C03652=1113.772,23.201,-52.779,179.827,6.837,149.312
C03653=1113.768,23.416,-52.792,179.828,6.841,149.313
C03654=1113.763,23.631,-52.805,179.828,6.845,149.313
C03655=1113.760,23.845,-52.819,179.829,6.848,149.314
C03656=1113.754,24.095,-52.833,179.830,6.853,149.315
C03657=1113.749,24.344,-52.848,179.831,6.857,149.315
C03658=1113.744,24.593,-52.864,179.832,6.861,149.316
C03659=1113.739,24.842,-52.879,179.833,6.866,149.317
C03660=1113.733,25.092,-52.894,179.833,6.869,149.317
C03661=1113.729,25.342,-52.909,179.834,6.874,149.318
C03662=1113.724,25.591,-52.925,179.835,6.878,149.319
C03663=1113.719,25.841,-52.940,179.836,6.883,149.320
C03664=1113.714,26.090,-52.955,179.837,6.887,149.320
C03665=1113.709,26.339,-52.971,179.838,6.891,149.321
C03666=1113.705,26.589,-52.986,179.838,6.895,149.322
C03667=1113.699,26.839,-53.001,179.839,6.900,149.322
C03668=1113.694,27.088,-53.016,179.840,6.904,149.323
C03669=1113.689,27.338,-53.032,179.841,6.908,149.324
C03670=1113.683,27.587,-53.047,179.842,6.913,149.324
C03671=1113.679,27.836,-53.062,179.843,6.917,149.325
C03672=1113.674,28.086,-53.078,179.844,6.922,149.326
C03673=1113.669,28.336,-53.094,179.844,6.925,149.327
C03674=1113.664,28.585,-53.109,179.845,6.929,149.327
C03675=1113.659,28.834,-53.124,179.846,6.934,149.328
C03676=1113.655,29.084,-53.140,179.847,6.938,149.329
C03677=1113.649,29.333,-53.155,179.848,6.943,149.329
C03678=1113.644,29.583,-53.171,179.849,6.947,149.330
C03679=1113.639,29.832,-53.186,179.849,6.951,149.331
C03680=1113.634,30.082,-53.202,179.850,6.955,149.331
C03681=1113.629,30.331,-53.218,179.851,6.959,149.332
C03682=1113.624,30.580,-53.233,179.852,6.964,149.333
C03683=1113.619,30.830,-53.248,179.853,6.968,149.334
C03684=1113.614,31.080,-53.264,179.854,6.973,149.334
C03685=1113.609,31.329,-53.280,179.855,6.976,149.335
C03686=1113.604,31.578,-53.295,179.856,6.980,149.336
C03687=1113.599,31.828,-53.310,179.857,6.985,149.336
C03688=1113.594,32.078,-53.326,179.858,6.989,149.337
C03689=1113.589,32.327,-53.341,179.859,6.993,149.338
C03690=1113.584,32.576,-53.357,179.860,6.998,149.338
C03691=1113.579,32.827,-53.373,179.860,7.001,149.339
C03692=1113.574,33.076,-53.388,179.861,7.005,149.339
C03693=1113.569,33.324,-53.404,179.862,7.010,149.340
C03694=1113.564,33.574,-53.420,179.864,7.014,149.341
C03695=1113.559,33.824,-53.436,179.865,7.018,149.341
C03696=1113.554,34.073,-53.451,179.866,7.023,149.342
C03697=1113.548,34.323,-53.467,179.866,7.026,149.343
C03698=1113.544,34.572,-53.482,179.867,7.030,149.343
C03699=1113.539,34.821,-53.498,179.868,7.035,149.344
C03700=1113.534,35.071,-53.514,179.869,7.039,149.345
C03701=1113.529,35.321,-53.530,179.870,7.043,149.345
C03702=1113.524,35.570,-53.546,179.871,7.048,149.346
C03703=1113.519,35.819,-53.561,179.872,7.051,149.347
C03704=1113.515,36.034,-53.574,179.873,7.056,149.347
C03705=1113.510,36.248,-53.588,179.874,7.059,149.348
C03706=1113.506,36.462,-53.602,179.874,7.062,149.348
C03707=1113.502,36.677,-53.615,179.875,7.066,149.349
C03708=1113.498,36.891,-53.629,179.876,7.070,149.350
C03709=1113.493,37.105,-53.643,179.877,7.073,149.350
C03710=1113.489,37.320,-53.656,179.878,7.076,149.351
C03711=1113.485,37.534,-53.670,179.879,7.081,149.351
C03712=1113.479,37.783,-53.686,179.879,7.084,149.352
C03713=1113.475,38.033,-53.702,179.881,7.088,149.352
C03714=1113.469,38.282,-53.718,179.882,7.092,149.353
C03715=1113.465,38.532,-53.733,179.883,7.097,149.354
C03716=1113.460,38.781,-53.750,179.884,7.101,149.354
C03717=1113.455,39.030,-53.765,179.885,7.105,149.355
C03718=1113.450,39.280,-53.781,179.885,7.109,149.356
C03719=1113.445,39.529,-53.798,179.887,7.113,149.356
C03720=1113.440,39.779,-53.814,179.888,7.117,149.357
C03721=1113.435,40.029,-53.829,179.889,7.122,149.358
C03722=1113.430,40.278,-53.846,179.890,7.126,149.358
C03723=1113.425,40.527,-53.861,179.891,7.130,149.359
C03724=1113.420,40.776,-53.878,179.892,7.133,149.359
C03725=1113.415,41.026,-53.894,179.893,7.138,149.360
C03726=1113.410,41.275,-53.910,179.894,7.142,149.361
C03727=1113.405,41.525,-53.926,179.895,7.146,149.361
C03728=1113.400,41.775,-53.941,179.896,7.150,149.362
C03729=1113.395,42.024,-53.958,179.898,7.155,149.362
C03730=1113.390,42.273,-53.974,179.898,7.158,149.363
C03731=1113.386,42.523,-53.990,179.899,7.162,149.364
C03732=1113.380,42.772,-54.006,179.900,7.167,149.364
C03733=1113.376,43.022,-54.023,179.902,7.171,149.365
C03734=1113.370,43.271,-54.038,179.903,7.175,149.365
C03735=1113.366,43.521,-54.055,179.903,7.178,149.366
C03736=1113.361,43.770,-54.071,179.904,7.183,149.367
C03737=1113.356,44.020,-54.087,179.905,7.187,149.367
C03738=1113.351,44.268,-54.103,179.907,7.191,149.368
C03739=1113.346,44.519,-54.119,179.908,7.195,149.368
C03740=1113.341,44.767,-54.136,179.909,7.200,149.369
C03741=1113.336,45.017,-54.152,179.910,7.203,149.370
C03742=1113.330,45.266,-54.169,179.911,7.207,149.370
C03743=1113.326,45.516,-54.185,179.912,7.211,149.371
C03744=1113.321,45.765,-54.201,179.913,7.216,149.371
C03745=1113.316,46.015,-54.217,179.914,7.220,149.372
C03746=1113.311,46.264,-54.234,179.916,7.224,149.373
C03747=1113.306,46.514,-54.250,179.916,7.227,149.373
C03748=1113.301,46.763,-54.266,179.917,7.232,149.374
C03749=1113.297,47.012,-54.283,179.919,7.236,149.374
C03750=1113.292,47.262,-54.299,179.920,7.240,149.375
C03751=1113.286,47.511,-54.316,179.921,7.244,149.376
C03752=1113.282,47.761,-54.332,179.923,7.248,149.376
C03753=1113.276,48.010,-54.348,179.923,7.252,149.377
C03754=1113.272,48.260,-54.364,179.924,7.256,149.377
C03755=1113.267,48.508,-54.381,179.925,7.260,149.378
C03756=1113.262,48.758,-54.397,179.927,7.264,149.378
C03757=1113.257,49.008,-54.414,179.928,7.268,149.379
C03758=1113.252,49.257,-54.430,179.929,7.271,149.379
C03759=1113.247,49.507,-54.447,179.930,7.276,149.380
C03760=1113.243,49.721,-54.461,179.932,7.280,149.381
C03761=1113.239,49.935,-54.475,179.932,7.283,149.381
C03762=1113.234,50.149,-54.489,179.933,7.286,149.382
C03763=1113.230,50.363,-54.504,179.934,7.289,149.382
C03764=1113.226,50.578,-54.518,179.935,7.293,149.383
C03765=1113.222,50.792,-54.532,179.936,7.297,149.383
C03766=1113.217,51.006,-54.547,179.937,7.300,149.384
C03767=1113.213,51.220,-54.561,179.938,7.304,149.384
C03768=1113.208,51.470,-54.577,179.939,7.308,149.385
C03769=1113.203,51.719,-54.593,179.940,7.311,149.385
C03770=1113.198,51.969,-54.611,179.941,7.316,149.386
C03771=1113.193,52.218,-54.627,179.943,7.320,149.386
C03772=1113.188,52.467,-54.644,179.944,7.324,149.387
C03773=1113.183,52.717,-54.661,179.945,7.328,149.388
C03774=1113.179,52.966,-54.677,179.947,7.332,149.388
C03775=1113.174,53.215,-54.694,179.947,7.336,149.389
C03776=1113.168,53.465,-54.711,179.948,7.340,149.389
C03777=1113.164,53.714,-54.728,179.950,7.344,149.390
C03778=1113.159,53.963,-54.744,179.951,7.348,149.390
C03779=1113.154,54.213,-54.761,179.953,7.352,149.391
C03780=1113.149,54.462,-54.778,179.954,7.356,149.391
C03781=1113.144,54.711,-54.794,179.955,7.359,149.392
C03782=1113.139,54.961,-54.812,179.956,7.364,149.392
C03783=1113.134,55.210,-54.828,179.957,7.368,149.393
C03784=1113.130,55.460,-54.845,179.958,7.372,149.394
C03785=1113.124,55.709,-54.862,179.960,7.376,149.394
C03786=1113.120,55.958,-54.878,179.961,7.380,149.395
C03787=1113.114,56.208,-54.896,179.961,7.384,149.395
C03788=1113.109,56.457,-54.912,179.963,7.388,149.396
C03789=1113.104,56.707,-54.929,179.964,7.392,149.396
C03790=1113.100,56.956,-54.946,179.966,7.396,149.397
C03791=1113.095,57.206,-54.963,179.967,7.400,149.397
C03792=1113.089,57.455,-54.980,179.968,7.404,149.398
C03793=1113.085,57.704,-54.996,179.969,7.408,149.399
C03794=1113.080,57.954,-55.013,179.970,7.411,149.399
C03795=1113.075,58.203,-55.031,179.971,7.416,149.400
C03796=1113.070,58.452,-55.048,179.973,7.420,149.400
C03797=1113.065,58.702,-55.064,179.974,7.424,149.401
C03798=1113.060,58.951,-55.082,179.976,7.428,149.401
C03799=1113.055,59.201,-55.098,179.977,7.432,149.402
C03800=1113.050,59.451,-55.116,179.978,7.436,149.402
C03801=1113.045,59.699,-55.133,179.979,7.439,149.403
C03802=1113.040,59.949,-55.150,179.980,7.443,149.403
C03803=1113.036,60.198,-55.167,179.982,7.447,149.404
C03804=1113.031,60.448,-55.184,179.983,7.452,149.404
C03805=1113.026,60.697,-55.201,179.985,7.456,149.405
C03806=1113.021,60.946,-55.218,179.986,7.460,149.405
C03807=1113.016,61.195,-55.235,179.987,7.464,149.406
C03808=1113.011,61.445,-55.252,179.988,7.467,149.407
C03809=1113.007,61.694,-55.269,179.989,7.471,149.407
C03810=1113.001,61.944,-55.287,179.991,7.475,149.407
C03811=1112.997,62.193,-55.303,179.992,7.479,149.408
C03812=1112.992,62.442,-55.321,179.994,7.483,149.409
C03813=1112.986,62.692,-55.338,179.995,7.488,149.409
C03814=1112.982,62.941,-55.355,179.996,7.491,149.410
C03815=1112.977,63.190,-55.373,179.997,7.495,149.410
C03816=1112.973,63.404,-55.387,179.998,7.499,149.411
C03817=1112.969,63.619,-55.403,179.999,7.502,149.411
C03818=1112.965,63.832,-55.417,-180.000,7.505,149.412
C03819=1112.960,64.047,-55.431,-179.998,7.509,149.412
C03820=1112.956,64.262,-55.447,-179.997,7.512,149.412
C03821=1112.952,64.475,-55.461,-179.996,7.515,149.413
C03822=1112.947,64.689,-55.476,-179.995,7.519,149.413
C03823=1112.943,64.904,-55.491,-179.994,7.522,149.414
C03824=1112.939,65.153,-55.509,-179.992,7.526,149.414
C03825=1112.933,65.403,-55.526,-179.991,7.530,149.415
C03826=1112.929,65.652,-55.544,-179.990,7.534,149.415
C03827=1112.924,65.901,-55.561,-179.988,7.538,149.416
C03828=1112.918,66.150,-55.579,-179.988,7.542,149.416
C03829=1112.914,66.399,-55.595,-179.986,7.546,149.417
C03830=1112.909,66.649,-55.613,-179.985,7.550,149.417
C03831=1112.904,66.898,-55.630,-179.983,7.554,149.418
C03832=1112.900,67.147,-55.648,-179.982,7.558,149.418
C03833=1112.894,67.397,-55.665,-179.981,7.562,149.419
C03834=1112.890,67.646,-55.683,-179.979,7.566,149.419
C03835=1112.884,67.896,-55.700,-179.978,7.570,149.420
C03836=1112.880,68.145,-55.718,-179.977,7.573,149.420
C03837=1112.875,68.395,-55.735,-179.975,7.577,149.421
C03838=1112.870,68.644,-55.753,-179.974,7.581,149.421
C03839=1112.865,68.893,-55.771,-179.973,7.585,149.422
C03840=1112.861,69.143,-55.788,-179.971,7.589,149.422
C03841=1112.856,69.392,-55.806,-179.970,7.593,149.423
C03842=1112.851,69.641,-55.824,-179.969,7.598,149.423
C03843=1112.846,69.891,-55.841,-179.967,7.601,149.424
C03844=1112.841,70.140,-55.859,-179.965,7.605,149.424
C03845=1112.836,70.389,-55.875,-179.964,7.610,149.425
C03846=1112.831,70.639,-55.893,-179.963,7.613,149.425
C03847=1112.826,70.888,-55.911,-179.962,7.617,149.426
C03848=1112.821,71.137,-55.929,-179.961,7.621,149.426
C03849=1112.816,71.387,-55.947,-179.959,7.625,149.427
C03850=1112.811,71.636,-55.965,-179.958,7.629,149.427
C03851=1112.807,71.885,-55.982,-179.956,7.633,149.428
C03852=1112.802,72.134,-55.999,-179.955,7.637,149.428
C03853=1112.797,72.384,-56.017,-179.953,7.641,149.429
C03854=1112.792,72.633,-56.035,-179.952,7.645,149.429
C03855=1112.787,72.882,-56.053,-179.951,7.649,149.430
C03856=1112.782,73.132,-56.071,-179.949,7.653,149.430
C03857=1112.777,73.381,-56.088,-179.948,7.656,149.431
C03858=1112.772,73.630,-56.106,-179.947,7.660,149.431
C03859=1112.767,73.879,-56.124,-179.945,7.664,149.432
C03860=1112.763,74.129,-56.143,-179.944,7.668,149.432
C03861=1112.759,74.378,-56.160,-179.942,7.672,149.433
C03862=1112.754,74.628,-56.177,-179.941,7.676,149.433
C03863=1112.749,74.877,-56.195,-179.939,7.680,149.434
C03864=1112.744,75.126,-56.213,-179.938,7.684,149.434
C03865=1112.739,75.375,-56.231,-179.937,7.688,149.435
C03866=1112.734,75.625,-56.249,-179.935,7.692,149.435
C03867=1112.729,75.874,-56.267,-179.934,7.696,149.436
C03868=1112.724,76.123,-56.285,-179.932,7.700,149.436
C03869=1112.719,76.372,-56.303,-179.931,7.704,149.437
C03870=1112.715,76.622,-56.322,-179.930,7.707,149.437
C03871=1112.710,76.872,-56.339,-179.928,7.711,149.438
C03872=1112.705,77.085,-56.355,-179.927,7.715,149.438
C03873=1112.701,77.300,-56.370,-179.927,7.718,149.439
C03874=1112.697,77.513,-56.386,-179.926,7.721,149.439
C03875=1112.693,77.728,-56.401,-179.925,7.724,149.440
C03876=1112.688,77.941,-56.417,-179.924,7.727,149.440
C03877=1112.685,78.156,-56.432,-179.923,7.730,149.441
C03878=1112.680,78.369,-56.447,-179.923,7.734,149.441
C03879=1112.676,78.584,-56.463,-179.922,7.737,149.442
C03880=1112.671,78.833,-56.481,-179.920,7.741,149.442
C03881=1112.666,79.082,-56.499,-179.920,7.744,149.443
C03882=1112.661,79.331,-56.517,-179.918,7.749,149.443
C03883=1112.656,79.582,-56.536,-179.917,7.752,149.444
C03884=1112.652,79.830,-56.554,-179.916,7.756,149.444
C03885=1112.647,80.079,-56.572,-179.915,7.759,149.445
C03886=1112.642,80.329,-56.590,-179.914,7.764,149.446
C03887=1112.637,80.578,-56.608,-179.913,7.767,149.446
C03888=1112.633,80.828,-56.627,-179.912,7.771,149.447
C03889=1112.628,81.077,-56.645,-179.911,7.774,149.447
C03890=1112.623,81.326,-56.663,-179.910,7.778,149.448
C03891=1112.618,81.575,-56.681,-179.909,7.781,149.448
C03892=1112.612,81.825,-56.699,-179.908,7.786,149.449
C03893=1112.608,82.075,-56.718,-179.906,7.790,149.449
C03894=1112.603,82.323,-56.736,-179.906,7.793,149.450
C03895=1112.599,82.572,-56.754,-179.904,7.797,149.450
C03896=1112.594,82.821,-56.772,-179.904,7.801,149.451
C03897=1112.589,83.071,-56.791,-179.902,7.804,149.451
C03898=1112.584,83.321,-56.809,-179.901,7.809,149.452
C03899=1112.579,83.569,-56.828,-179.900,7.812,149.452
C03900=1112.574,83.818,-56.846,-179.899,7.816,149.453
C03901=1112.570,84.068,-56.864,-179.898,7.819,149.453
C03902=1112.565,84.318,-56.882,-179.896,7.823,149.454
C03903=1112.560,84.567,-56.900,-179.895,7.827,149.455
C03904=1112.555,84.816,-56.919,-179.894,7.830,149.455
C03905=1112.550,85.065,-56.938,-179.893,7.835,149.456
C03906=1112.545,85.315,-56.956,-179.892,7.839,149.456
C03907=1112.540,85.564,-56.974,-179.891,7.842,149.457
C03908=1112.535,85.813,-56.993,-179.889,7.846,149.457
C03909=1112.531,86.063,-57.011,-179.888,7.850,149.458
C03910=1112.526,86.312,-57.029,-179.887,7.853,149.458
C03911=1112.521,86.560,-57.048,-179.886,7.857,149.459
C03912=1112.516,86.810,-57.067,-179.884,7.861,149.459
C03913=1112.511,87.060,-57.085,-179.884,7.865,149.460
C03914=1112.507,87.308,-57.104,-179.882,7.869,149.460
C03915=1112.502,87.558,-57.123,-179.881,7.872,149.461
C03916=1112.497,87.808,-57.141,-179.880,7.876,149.461
C03917=1112.492,88.056,-57.159,-179.878,7.880,149.462
C03918=1112.487,88.306,-57.178,-179.877,7.884,149.462
C03919=1112.483,88.555,-57.197,-179.876,7.888,149.463
C03920=1112.478,88.804,-57.215,-179.875,7.891,149.463
C03921=1112.473,89.054,-57.233,-179.873,7.895,149.464
C03922=1112.468,89.303,-57.252,-179.872,7.899,149.464
C03923=1112.463,89.552,-57.270,-179.870,7.903,149.465
C03924=1112.458,89.802,-57.290,-179.869,7.906,149.465
C03925=1112.453,90.051,-57.308,-179.868,7.911,149.466
C03926=1112.449,90.299,-57.327,-179.867,7.914,149.466
C03927=1112.444,90.549,-57.346,-179.865,7.918,149.467
C03928=1112.439,90.763,-57.361,-179.864,7.921,149.467
C03929=1112.436,90.977,-57.378,-179.863,7.925,149.468
C03930=1112.432,91.191,-57.394,-179.862,7.928,149.468
C03931=1112.428,91.405,-57.410,-179.861,7.932,149.468
C03932=1112.423,91.619,-57.425,-179.860,7.935,149.469
C03933=1112.419,91.833,-57.442,-179.858,7.937,149.469
C03934=1112.415,92.047,-57.458,-179.857,7.941,149.469
C03935=1112.411,92.260,-57.474,-179.856,7.944,149.470
C03936=1112.406,92.510,-57.494,-179.854,7.948,149.470
C03937=1112.401,92.759,-57.512,-179.853,7.952,149.471
C03938=1112.397,93.008,-57.531,-179.852,7.956,149.471
C03939=1112.391,93.258,-57.549,-179.850,7.960,149.472
C03940=1112.387,93.506,-57.568,-179.849,7.963,149.472
C03941=1112.382,93.756,-57.588,-179.847,7.967,149.473
C03942=1112.377,94.005,-57.606,-179.846,7.971,149.473
C03943=1112.372,94.255,-57.625,-179.845,7.974,149.474
C03944=1112.367,94.504,-57.643,-179.843,7.978,149.474
C03945=1112.363,94.754,-57.663,-179.841,7.982,149.474
C03946=1112.358,95.002,-57.682,-179.840,7.986,149.475
C03947=1112.353,95.252,-57.701,-179.839,7.990,149.476
C03948=1112.348,95.501,-57.719,-179.837,7.994,149.476
C03949=1112.343,95.750,-57.739,-179.835,7.998,149.476
C03950=1112.339,95.999,-57.758,-179.834,8.001,149.477
C03951=1112.333,96.248,-57.776,-179.833,8.005,149.477
C03952=1112.329,96.498,-57.796,-179.831,8.009,149.478
C03953=1112.324,96.747,-57.815,-179.830,8.013,149.478
C03954=1112.319,96.996,-57.834,-179.828,8.017,149.479
C03955=1112.314,97.245,-57.852,-179.826,8.021,149.479
C03956=1112.310,97.495,-57.872,-179.825,8.025,149.479
C03957=1112.305,97.743,-57.891,-179.823,8.028,149.480
C03958=1112.300,97.993,-57.910,-179.821,8.032,149.480
C03959=1112.295,98.242,-57.929,-179.820,8.036,149.481
C03960=1112.291,98.492,-57.948,-179.818,8.040,149.481
C03961=1112.286,98.741,-57.967,-179.816,8.044,149.481
C03962=1112.281,98.990,-57.986,-179.815,8.047,149.482
C03963=1112.277,99.239,-58.006,-179.814,8.051,149.482
C03964=1112.271,99.488,-58.025,-179.812,8.054,149.483
C03965=1112.267,99.738,-58.044,-179.811,8.058,149.483
C03966=1112.262,99.986,-58.063,-179.809,8.062,149.483
C03967=1112.257,100.236,-58.083,-179.807,8.066,149.484
C03968=1112.252,100.485,-58.101,-179.805,8.070,149.484
C03969=1112.247,100.735,-58.121,-179.804,8.074,149.485
C03970=1112.243,100.984,-58.140,-179.802,8.077,149.485
C03971=1112.237,101.233,-58.160,-179.800,8.081,149.485
C03972=1112.233,101.482,-58.179,-179.798,8.085,149.486
C03973=1112.228,101.731,-58.198,-179.797,8.089,149.486
C03974=1112.223,101.981,-58.218,-179.795,8.093,149.487
C03975=1112.219,102.229,-58.236,-179.793,8.096,149.487
C03976=1112.214,102.479,-58.256,-179.792,8.100,149.487
C03977=1112.209,102.729,-58.276,-179.790,8.104,149.488
C03978=1112.204,102.977,-58.295,-179.788,8.107,149.488
C03979=1112.200,103.227,-58.314,-179.786,8.111,149.488
C03980=1112.195,103.476,-58.334,-179.785,8.115,149.489
C03981=1112.190,103.725,-58.354,-179.783,8.119,149.489
C03982=1112.185,103.974,-58.373,-179.781,8.122,149.489
C03983=1112.180,104.223,-58.393,-179.779,8.126,149.490
C03984=1112.176,104.437,-58.409,-179.777,8.130,149.490
C03985=1112.172,104.651,-58.426,-179.776,8.133,149.490
C03986=1112.168,104.865,-58.442,-179.775,8.136,149.491
C03987=1112.164,105.079,-58.460,-179.773,8.139,149.491
C03988=1112.160,105.293,-58.476,-179.772,8.142,149.491
C03989=1112.156,105.507,-58.493,-179.769,8.145,149.491
C03990=1112.152,105.721,-58.509,-179.768,8.149,149.492
C03991=1112.148,105.934,-58.527,-179.766,8.152,149.492
C03992=1112.142,106.183,-58.546,-179.765,8.156,149.493
C03993=1112.138,106.433,-58.565,-179.763,8.159,149.493
C03994=1112.134,106.682,-58.585,-179.761,8.163,149.493
C03995=1112.129,106.931,-58.605,-179.759,8.167,149.493
C03996=1112.124,107.180,-58.624,-179.757,8.170,149.494
C03997=1112.119,107.430,-58.644,-179.755,8.174,149.494
C03998=1112.115,107.679,-58.664,-179.753,8.178,149.494
C03999=1112.109,107.927,-58.684,-179.751,8.181,149.495
C04000=1112.105,108.177,-58.703,-179.750,8.185,149.495
C04001=1112.100,108.427,-58.723,-179.748,8.189,149.495
C04002=1112.095,108.675,-58.743,-179.745,8.193,149.495
C04003=1112.090,108.924,-58.763,-179.743,8.197,149.496
C04004=1112.086,109.174,-58.782,-179.741,8.200,149.496
C04005=1112.082,109.423,-58.802,-179.739,8.204,149.496
C04006=1112.077,109.672,-58.822,-179.738,8.208,149.497
C04007=1112.072,109.921,-58.841,-179.736,8.211,149.497
C04008=1112.067,110.170,-58.861,-179.734,8.215,149.497
C04009=1112.062,110.419,-58.881,-179.731,8.218,149.497
C04010=1112.058,110.668,-58.901,-179.729,8.222,149.498
C04011=1112.053,110.917,-58.921,-179.728,8.226,149.498
C04012=1112.048,111.167,-58.940,-179.726,8.229,149.498
C04013=1112.043,111.416,-58.961,-179.724,8.233,149.499
C04014=1112.038,111.666,-58.981,-179.722,8.236,149.499
C04015=1112.033,111.915,-59.001,-179.720,8.240,149.499
C04016=1112.028,112.164,-59.021,-179.719,8.243,149.499
C04017=1112.024,112.412,-59.041,-179.717,8.247,149.500
C04018=1112.019,112.662,-59.061,-179.715,8.250,149.500
C04019=1112.015,112.911,-59.081,-179.713,8.254,149.500
C04020=1112.010,113.161,-59.101,-179.711,8.257,149.501
C04021=1112.005,113.410,-59.121,-179.710,8.260,149.501
C04022=1112.000,113.658,-59.140,-179.708,8.264,149.501
C04023=1111.996,113.907,-59.161,-179.706,8.268,149.502
C04024=1111.991,114.157,-59.180,-179.704,8.271,149.502
C04025=1111.986,114.406,-59.201,-179.703,8.274,149.502
C04026=1111.981,114.655,-59.222,-179.701,8.278,149.503
C04027=1111.976,114.905,-59.241,-179.699,8.281,149.503
C04028=1111.971,115.153,-59.261,-179.697,8.285,149.503
C04029=1111.967,115.402,-59.281,-179.695,8.287,149.503
C04030=1111.962,115.651,-59.301,-179.694,8.291,149.504
C04031=1111.958,115.900,-59.322,-179.692,8.295,149.504
C04032=1111.952,116.150,-59.342,-179.690,8.298,149.504
C04033=1111.948,116.399,-59.362,-179.689,8.301,149.505
C04034=1111.943,116.648,-59.383,-179.687,8.305,149.505
C04035=1111.939,116.898,-59.402,-179.685,8.308,149.505
C04036=1111.934,117.147,-59.423,-179.683,8.311,149.505
C04037=1111.928,117.395,-59.443,-179.682,8.315,149.506
C04038=1111.924,117.644,-59.464,-179.679,8.318,149.506
C04039=1111.919,117.894,-59.483,-179.677,8.322,149.506
C04040=1111.915,118.108,-59.501,-179.676,8.325,149.506
C04041=1111.911,118.322,-59.519,-179.675,8.327,149.507
C04042=1111.907,118.535,-59.537,-179.674,8.330,149.507
C04043=1111.903,118.749,-59.554,-179.672,8.333,149.507
C04044=1111.900,118.962,-59.571,-179.670,8.337,149.507
C04045=1111.895,119.176,-59.588,-179.669,8.339,149.508
C04046=1111.891,119.390,-59.606,-179.667,8.342,149.508
C04047=1111.887,119.604,-59.623,-179.666,8.345,149.508
C04048=1111.882,119.853,-59.644,-179.664,8.348,149.508
C04049=1111.877,120.102,-59.665,-179.662,8.352,149.509
C04050=1111.873,120.351,-59.685,-179.661,8.355,149.509
C04051=1111.868,120.600,-59.705,-179.659,8.358,149.509
C04052=1111.863,120.850,-59.726,-179.656,8.362,149.509
C04053=1111.859,121.099,-59.746,-179.655,8.365,149.510
C04054=1111.854,121.348,-59.766,-179.653,8.368,149.510
C04055=1111.849,121.597,-59.787,-179.651,8.372,149.510
C04056=1111.844,121.846,-59.808,-179.650,8.375,149.511
C04057=1111.840,122.095,-59.828,-179.648,8.378,149.511
C04058=1111.835,122.344,-59.849,-179.646,8.382,149.511
C04059=1111.830,122.593,-59.869,-179.644,8.386,149.511
C04060=1111.826,122.842,-59.890,-179.643,8.388,149.512
C04061=1111.821,123.091,-59.911,-179.641,8.392,149.512
C04062=1111.816,123.340,-59.931,-179.639,8.396,149.512
C04063=1111.812,123.589,-59.951,-179.638,8.398,149.513
C04064=1111.807,123.838,-59.972,-179.636,8.402,149.513
C04065=1111.802,124.087,-59.993,-179.633,8.405,149.513
C04066=1111.797,124.337,-60.014,-179.632,8.408,149.513
C04067=1111.793,124.586,-60.034,-179.630,8.412,149.514
C04068=1111.788,124.836,-60.055,-179.628,8.415,149.514
C04069=1111.784,125.084,-60.076,-179.627,8.418,149.514
C04070=1111.779,125.333,-60.096,-179.625,8.422,149.515
C04071=1111.774,125.583,-60.117,-179.623,8.426,149.515
C04072=1111.770,125.832,-60.138,-179.621,8.429,149.515
C04073=1111.764,126.081,-60.159,-179.620,8.432,149.515
C04074=1111.760,126.330,-60.179,-179.618,8.436,149.516
C04075=1111.755,126.579,-60.200,-179.616,8.439,149.516
C04076=1111.750,126.828,-60.220,-179.615,8.442,149.516
C04077=1111.746,127.077,-60.242,-179.613,8.445,149.516
C04078=1111.741,127.326,-60.262,-179.610,8.449,149.517
C04079=1111.737,127.576,-60.284,-179.609,8.452,149.517
C04080=1111.732,127.825,-60.304,-179.607,8.455,149.517
C04081=1111.727,128.074,-60.325,-179.605,8.459,149.518
C04082=1111.723,128.323,-60.345,-179.604,8.462,149.518
C04083=1111.718,128.571,-60.367,-179.602,8.466,149.518
C04084=1111.713,128.820,-60.387,-179.600,8.469,149.518
C04085=1111.708,129.070,-60.408,-179.599,8.472,149.519
C04086=1111.703,129.319,-60.429,-179.597,8.475,149.519
C04087=1111.699,129.568,-60.451,-179.595,8.479,149.519
C04088=1111.694,129.817,-60.472,-179.594,8.482,149.520
C04089=1111.690,130.066,-60.492,-179.592,8.485,149.520
C04090=1111.685,130.315,-60.513,-179.589,8.489,149.520
C04091=1111.680,130.564,-60.535,-179.588,8.492,149.520
C04092=1111.675,130.813,-60.555,-179.586,8.495,149.521
C04093=1111.671,131.063,-60.576,-179.584,8.499,149.521
C04094=1111.667,131.311,-60.598,-179.583,8.502,149.521
C04095=1111.661,131.561,-60.619,-179.581,8.505,149.522
C04096=1111.657,131.774,-60.637,-179.580,8.508,149.522
C04097=1111.652,131.988,-60.655,-179.578,8.511,149.522
C04098=1111.649,132.202,-60.673,-179.576,8.514,149.522
C04099=1111.645,132.415,-60.691,-179.575,8.517,149.522
C04100=1111.641,132.629,-60.709,-179.573,8.520,149.523
C04101=1111.638,132.842,-60.727,-179.572,8.523,149.523
C04102=1111.633,133.056,-60.746,-179.571,8.525,149.523
C04103=1111.629,133.270,-60.763,-179.570,8.528,149.524
C04104=1111.624,133.519,-60.785,-179.567,8.532,149.524
C04105=1111.620,133.768,-60.806,-179.565,8.535,149.524
C04106=1111.615,134.017,-60.827,-179.564,8.538,149.524
C04107=1111.610,134.266,-60.848,-179.562,8.542,149.525
C04108=1111.605,134.515,-60.869,-179.560,8.545,149.525
C04109=1111.601,134.764,-60.891,-179.559,8.548,149.525
C04110=1111.596,135.013,-60.912,-179.557,8.552,149.526
C04111=1111.591,135.262,-60.933,-179.555,8.555,149.526
C04112=1111.587,135.511,-60.954,-179.554,8.558,149.526
C04113=1111.582,135.760,-60.976,-179.552,8.562,149.527
C04114=1111.577,136.010,-60.997,-179.550,8.566,149.527
C04115=1111.572,136.258,-61.019,-179.548,8.568,149.527
C04116=1111.569,136.507,-61.040,-179.547,8.572,149.527
C04117=1111.564,136.757,-61.061,-179.545,8.576,149.528
C04118=1111.559,137.005,-61.083,-179.543,8.578,149.528
C04119=1111.554,137.254,-61.104,-179.542,8.582,149.528
C04120=1111.549,137.504,-61.126,-179.540,8.586,149.529
C04121=1111.545,137.752,-61.147,-179.538,8.588,149.529
C04122=1111.540,138.001,-61.168,-179.537,8.592,149.529
C04123=1111.536,138.251,-61.190,-179.534,8.596,149.529
C04124=1111.531,138.500,-61.211,-179.533,8.599,149.530
C04125=1111.526,138.749,-61.232,-179.531,8.602,149.530
C04126=1111.521,138.998,-61.254,-179.529,8.606,149.530
C04127=1111.517,139.247,-61.275,-179.528,8.609,149.531
C04128=1111.512,139.496,-61.296,-179.526,8.612,149.531
C04129=1111.508,139.745,-61.319,-179.524,8.616,149.531
C04130=1111.503,139.994,-61.340,-179.523,8.619,149.532
C04131=1111.498,140.243,-61.361,-179.521,8.623,149.532
C04132=1111.494,140.492,-61.383,-179.519,8.626,149.532
C04133=1111.489,140.741,-61.405,-179.518,8.629,149.533
C04134=1111.484,140.990,-61.426,-179.516,8.633,149.533
C04135=1111.479,141.239,-61.448,-179.514,8.636,149.533
C04136=1111.475,141.488,-61.469,-179.512,8.640,149.534
C04137=1111.471,141.737,-61.491,-179.511,8.643,149.534
C04138=1111.466,141.986,-61.513,-179.509,8.647,149.534
C04139=1111.461,142.235,-61.534,-179.507,8.650,149.534
C04140=1111.457,142.484,-61.556,-179.506,8.653,149.535
C04141=1111.452,142.733,-61.577,-179.504,8.657,149.535
C04142=1111.447,142.982,-61.599,-179.502,8.660,149.536
C04143=1111.443,143.231,-61.621,-179.501,8.663,149.536
C04144=1111.438,143.480,-61.643,-179.499,8.667,149.536
C04145=1111.433,143.730,-61.664,-179.497,8.671,149.536
C04146=1111.428,143.978,-61.686,-179.496,8.674,149.537
C04147=1111.424,144.228,-61.708,-179.494,8.677,149.537
C04148=1111.419,144.476,-61.730,-179.492,8.681,149.538
C04149=1111.415,144.726,-61.752,-179.490,8.684,149.538
C04150=1111.410,144.974,-61.773,-179.489,8.688,149.538
C04151=1111.405,145.223,-61.795,-179.487,8.691,149.538
C04152=1111.401,145.437,-61.814,-179.486,8.694,149.539
C04153=1111.397,145.650,-61.832,-179.484,8.697,149.539
C04154=1111.393,145.864,-61.851,-179.482,8.700,149.539
C04155=1111.389,146.077,-61.870,-179.480,8.703,149.539
C04156=1111.385,146.291,-61.889,-179.479,8.706,149.540
C04157=1111.381,146.504,-61.907,-179.477,8.710,149.540
C04158=1111.377,146.718,-61.926,-179.475,8.712,149.540
C04159=1111.374,146.931,-61.945,-179.473,8.716,149.540
C04160=1111.369,147.181,-61.968,-179.472,8.720,149.541
C04161=1111.364,147.429,-61.990,-179.469,8.723,149.541
C04162=1111.359,147.679,-62.012,-179.467,8.727,149.541
C04163=1111.355,147.927,-62.033,-179.465,8.730,149.541
C04164=1111.350,148.177,-62.055,-179.463,8.734,149.542
C04165=1111.345,148.425,-62.077,-179.461,8.737,149.542
C04166=1111.341,148.675,-62.099,-179.459,8.741,149.542
C04167=1111.336,148.923,-62.121,-179.457,8.744,149.542
C04168=1111.331,149.173,-62.143,-179.455,8.748,149.543
C04169=1111.327,149.422,-62.165,-179.453,8.751,149.543
C04170=1111.322,149.670,-62.188,-179.451,8.755,149.543
C04171=1111.318,149.920,-62.210,-179.449,8.758,149.543
C04172=1111.313,150.168,-62.232,-179.447,8.762,149.544
C04173=1111.308,150.418,-62.254,-179.444,8.765,149.544
C04174=1111.303,150.666,-62.276,-179.442,8.769,149.544
C04175=1111.299,150.915,-62.299,-179.440,8.772,149.544
C04176=1111.295,151.164,-62.320,-179.438,8.776,149.545
C04177=1111.290,151.413,-62.343,-179.436,8.779,149.545
C04178=1111.285,151.663,-62.365,-179.434,8.783,149.545
C04179=1111.280,151.911,-62.387,-179.432,8.786,149.545
C04180=1111.276,152.160,-62.410,-179.430,8.789,149.545
C04181=1111.271,152.409,-62.432,-179.427,8.793,149.546
C04182=1111.267,152.658,-62.454,-179.425,8.796,149.546
C04183=1111.262,152.906,-62.476,-179.423,8.800,149.546
C04184=1111.257,153.156,-62.499,-179.421,8.803,149.546
C04185=1111.253,153.405,-62.521,-179.419,8.807,149.546
C04186=1111.248,153.653,-62.543,-179.417,8.810,149.547
C04187=1111.243,153.903,-62.566,-179.414,8.813,149.547
C04188=1111.239,154.152,-62.588,-179.413,8.816,149.547
C04189=1111.234,154.401,-62.610,-179.411,8.819,149.547
C04190=1111.229,154.650,-62.633,-179.409,8.823,149.547
C04191=1111.225,154.898,-62.655,-179.406,8.826,149.547
C04192=1111.221,155.148,-62.678,-179.404,8.829,149.548
C04193=1111.216,155.397,-62.701,-179.402,8.833,149.548
C04194=1111.211,155.645,-62.723,-179.400,8.836,149.548
C04195=1111.206,155.895,-62.745,-179.398,8.840,149.548
C04196=1111.202,156.144,-62.768,-179.395,8.843,149.548
C04197=1111.197,156.392,-62.790,-179.394,8.846,149.549
C04198=1111.192,156.641,-62.813,-179.391,8.849,149.549
C04199=1111.188,156.891,-62.835,-179.389,8.852,149.549
C04200=1111.183,157.140,-62.858,-179.387,8.856,149.549
C04201=1111.179,157.388,-62.880,-179.385,8.859,149.549
C04202=1111.175,157.637,-62.903,-179.383,8.862,149.549
C04203=1111.170,157.886,-62.926,-179.381,8.866,149.550
C04204=1111.165,158.135,-62.948,-179.379,8.868,149.550
C04205=1111.160,158.384,-62.971,-179.377,8.872,149.550
C04206=1111.156,158.633,-62.993,-179.375,8.875,149.550
C04207=1111.151,158.882,-63.017,-179.372,8.878,149.550
C04208=1111.147,159.095,-63.036,-179.371,8.881,149.551
C04209=1111.143,159.309,-63.055,-179.369,8.883,149.551
C04210=1111.140,159.522,-63.074,-179.367,8.887,149.551
C04211=1111.136,159.735,-63.094,-179.365,8.889,149.551
C04212=1111.132,159.949,-63.114,-179.363,8.892,149.551
C04213=1111.128,160.162,-63.133,-179.361,8.895,149.551
C04214=1111.124,160.376,-63.153,-179.359,8.898,149.551
C04215=1111.120,160.589,-63.172,-179.357,8.900,149.551
C04216=1111.115,160.838,-63.195,-179.355,8.903,149.552
C04217=1111.111,161.087,-63.218,-179.353,8.907,149.552
C04218=1111.106,161.337,-63.241,-179.351,8.909,149.552
C04219=1111.101,161.585,-63.263,-179.349,8.912,149.552
C04220=1111.097,161.834,-63.286,-179.347,8.916,149.552
C04221=1111.093,162.083,-63.309,-179.344,8.919,149.552
C04222=1111.088,162.332,-63.332,-179.342,8.923,149.552
C04223=1111.083,162.581,-63.355,-179.340,8.925,149.552
C04224=1111.078,162.829,-63.378,-179.338,8.928,149.553
C04225=1111.074,163.078,-63.401,-179.336,8.931,149.553
C04226=1111.070,163.327,-63.424,-179.334,8.935,149.553
C04227=1111.065,163.577,-63.446,-179.332,8.937,149.553
C04228=1111.060,163.826,-63.470,-179.330,8.941,149.553
C04229=1111.056,164.074,-63.493,-179.327,8.944,149.553
C04230=1111.051,164.323,-63.516,-179.325,8.947,149.553
C04231=1111.046,164.572,-63.539,-179.323,8.950,149.554
C04232=1111.042,164.820,-63.562,-179.321,8.953,149.554
C04233=1111.037,165.069,-63.585,-179.318,8.956,149.554
C04234=1111.033,165.319,-63.608,-179.316,8.959,149.554
C04235=1111.029,165.567,-63.631,-179.315,8.962,149.554
C04236=1111.024,165.816,-63.655,-179.312,8.965,149.554
C04237=1111.019,166.066,-63.677,-179.309,8.968,149.554
C04238=1111.014,166.314,-63.700,-179.307,8.972,149.554
C04239=1111.010,166.563,-63.723,-179.305,8.974,149.554
C04240=1111.005,166.812,-63.746,-179.303,8.978,149.555
C04241=1111.000,167.061,-63.770,-179.301,8.981,149.555
C04242=1110.996,167.310,-63.792,-179.299,8.983,149.555
C04243=1110.992,167.559,-63.816,-179.297,8.987,149.555
C04244=1110.987,167.808,-63.839,-179.294,8.990,149.555
C04245=1110.982,168.057,-63.862,-179.292,8.993,149.555
C04246=1110.978,168.305,-63.887,-179.290,8.995,149.555
C04247=1110.973,168.553,-63.909,-179.288,8.999,149.555
C04248=1110.969,168.802,-63.932,-179.286,9.002,149.556
C04249=1110.964,169.051,-63.956,-179.284,9.004,149.556
C04250=1110.959,169.300,-63.979,-179.281,9.007,149.556
C04251=1110.955,169.549,-64.002,-179.279,9.011,149.556
C04252=1110.951,169.798,-64.025,-179.277,9.014,149.556
C04253=1110.946,170.047,-64.048,-179.275,9.016,149.556
C04254=1110.941,170.296,-64.072,-179.273,9.020,149.556
C04255=1110.937,170.545,-64.096,-179.270,9.023,149.556
C04256=1110.932,170.794,-64.119,-179.268,9.025,149.556
C04257=1110.927,171.043,-64.143,-179.266,9.029,149.556
C04258=1110.923,171.292,-64.166,-179.264,9.032,149.557
C04259=1110.918,171.541,-64.189,-179.262,9.034,149.557
C04260=1110.914,171.789,-64.213,-179.260,9.038,149.557
C04261=1110.910,172.038,-64.236,-179.257,9.041,149.557
C04262=1110.905,172.287,-64.260,-179.255,9.043,149.557
C04263=1110.900,172.536,-64.283,-179.253,9.047,149.557
C04264=1110.897,172.749,-64.303,-179.251,9.049,149.557
C04265=1110.892,172.963,-64.324,-179.250,9.051,149.557
C04266=1110.888,173.176,-64.344,-179.248,9.054,149.557
C04267=1110.885,173.389,-64.364,-179.246,9.057,149.557
C04268=1110.881,173.602,-64.384,-179.244,9.059,149.558
C04269=1110.876,173.816,-64.404,-179.242,9.062,149.558
C04270=1110.873,174.029,-64.425,-179.240,9.065,149.558
C04271=1110.869,174.242,-64.444,-179.238,9.067,149.558
C04272=1110.864,174.491,-64.468,-179.236,9.070,149.558
C04273=1110.860,174.740,-64.492,-179.234,9.073,149.558
C04274=1110.855,174.989,-64.515,-179.232,9.076,149.558
C04275=1110.851,175.237,-64.539,-179.229,9.079,149.558
C04276=1110.847,175.487,-64.563,-179.228,9.082,149.558
C04277=1110.842,175.736,-64.587,-179.225,9.085,149.558
C04278=1110.837,175.985,-64.610,-179.223,9.088,149.558
C04279=1110.833,176.234,-64.634,-179.221,9.090,149.559
C04280=1110.828,176.482,-64.658,-179.219,9.094,149.559
C04281=1110.824,176.731,-64.681,-179.216,9.097,149.559
C04282=1110.819,176.979,-64.705,-179.214,9.099,149.559
C04283=1110.815,177.228,-64.729,-179.212,9.103,149.559
C04284=1110.810,177.477,-64.753,-179.210,9.106,149.559
C04285=1110.805,177.726,-64.777,-179.208,9.108,149.559
C04286=1110.801,177.975,-64.801,-179.206,9.111,149.559
C04287=1110.796,178.224,-64.824,-179.203,9.115,149.559
C04288=1110.792,178.473,-64.848,-179.201,9.117,149.559
C04289=1110.787,178.722,-64.872,-179.199,9.120,149.560
C04290=1110.783,178.970,-64.896,-179.197,9.124,149.560
C04291=1110.778,179.219,-64.919,-179.195,9.126,149.560
C04292=1110.774,179.468,-64.943,-179.193,9.129,149.560
C04293=1110.769,179.716,-64.967,-179.190,9.132,149.560
C04294=1110.764,179.966,-64.992,-179.188,9.136,149.560
C04295=1110.760,180.215,-65.016,-179.185,9.139,149.560
C04296=1110.756,180.463,-65.040,-179.183,9.142,149.560
C04297=1110.751,180.712,-65.063,-179.181,9.144,149.560
C04298=1110.747,180.960,-65.087,-179.178,9.147,149.560
C04299=1110.743,181.210,-65.112,-179.176,9.150,149.560
C04300=1110.737,181.459,-65.136,-179.174,9.154,149.561
C04301=1110.733,181.707,-65.160,-179.171,9.157,149.561
C04302=1110.729,181.956,-65.184,-179.169,9.160,149.561
C04303=1110.724,182.205,-65.207,-179.167,9.162,149.561
C04304=1110.720,182.454,-65.232,-179.164,9.165,149.561
C04305=1110.715,182.703,-65.256,-179.162,9.169,149.561
C04306=1110.711,182.951,-65.280,-179.159,9.172,149.561
C04307=1110.706,183.200,-65.304,-179.157,9.174,149.561
C04308=1110.701,183.448,-65.328,-179.155,9.177,149.561
C04309=1110.697,183.698,-65.353,-179.152,9.180,149.561
C04310=1110.693,183.946,-65.377,-179.150,9.183,149.561
C04311=1110.688,184.195,-65.401,-179.148,9.186,149.561
C04312=1110.683,184.444,-65.425,-179.145,9.189,149.561
C04313=1110.679,184.693,-65.449,-179.143,9.192,149.561
C04314=1110.674,184.942,-65.473,-179.140,9.195,149.561
C04315=1110.670,185.190,-65.498,-179.138,9.197,149.561
C04316=1110.665,185.439,-65.522,-179.136,9.200,149.561
C04317=1110.661,185.688,-65.547,-179.133,9.204,149.561
C04318=1110.657,185.936,-65.571,-179.131,9.206,149.561
C04319=1110.652,186.185,-65.595,-179.129,9.209,149.561
C04320=1110.648,186.398,-65.615,-179.127,9.211,149.561
C04321=1110.644,186.612,-65.636,-179.125,9.213,149.561
C04322=1110.640,186.826,-65.658,-179.123,9.216,149.561
C04323=1110.637,187.039,-65.678,-179.120,9.219,149.561
C04324=1110.632,187.252,-65.699,-179.118,9.221,149.561
C04325=1110.629,187.465,-65.720,-179.117,9.223,149.561
C04326=1110.625,187.678,-65.741,-179.115,9.226,149.561
C04327=1110.621,187.891,-65.762,-179.113,9.228,149.562
C04328=1110.617,188.140,-65.787,-179.110,9.231,149.562
C04329=1110.612,188.389,-65.811,-179.108,9.234,149.562
C04330=1110.607,188.638,-65.835,-179.106,9.237,149.562
C04331=1110.602,188.886,-65.860,-179.103,9.240,149.562
C04332=1110.598,189.135,-65.884,-179.101,9.242,149.562
C04333=1110.594,189.384,-65.909,-179.099,9.245,149.562
C04334=1110.589,189.633,-65.933,-179.097,9.247,149.562
C04335=1110.585,189.881,-65.958,-179.094,9.251,149.562
C04336=1110.580,190.130,-65.983,-179.092,9.254,149.562
C04337=1110.576,190.379,-66.007,-179.090,9.256,149.562
C04338=1110.571,190.628,-66.032,-179.088,9.259,149.562
C04339=1110.567,190.876,-66.056,-179.086,9.261,149.562
C04340=1110.562,191.125,-66.081,-179.083,9.265,149.562
C04341=1110.558,191.374,-66.105,-179.081,9.267,149.562
C04342=1110.553,191.623,-66.130,-179.079,9.270,149.562
C04343=1110.549,191.871,-66.155,-179.077,9.274,149.562
C04344=1110.544,192.120,-66.180,-179.075,9.276,149.562
C04345=1110.540,192.369,-66.205,-179.072,9.279,149.563
C04346=1110.535,192.618,-66.229,-179.070,9.281,149.563
C04347=1110.530,192.866,-66.254,-179.068,9.284,149.563
C04348=1110.527,193.115,-66.279,-179.066,9.287,149.563
C04349=1110.521,193.364,-66.303,-179.063,9.290,149.563
C04350=1110.518,193.613,-66.328,-179.061,9.292,149.563
C04351=1110.513,193.861,-66.353,-179.059,9.296,149.563
C04352=1110.508,194.110,-66.378,-179.057,9.298,149.563
C04353=1110.504,194.359,-66.402,-179.055,9.301,149.563
C04354=1110.499,194.607,-66.427,-179.052,9.304,149.563
C04355=1110.495,194.856,-66.452,-179.051,9.307,149.563
C04356=1110.490,195.105,-66.477,-179.048,9.310,149.563
C04357=1110.486,195.354,-66.502,-179.047,9.312,149.563
C04358=1110.482,195.602,-66.527,-179.044,9.315,149.564
C04359=1110.477,195.851,-66.552,-179.042,9.318,149.564
C04360=1110.472,196.099,-66.577,-179.040,9.321,149.564
C04361=1110.468,196.348,-66.602,-179.038,9.324,149.564
C04362=1110.463,196.597,-66.626,-179.036,9.327,149.564
C04363=1110.459,196.846,-66.652,-179.033,9.330,149.564
C04364=1110.455,197.094,-66.676,-179.031,9.333,149.564
C04365=1110.450,197.343,-66.702,-179.028,9.336,149.564
C04366=1110.445,197.592,-66.726,-179.026,9.339,149.564
C04367=1110.442,197.840,-66.752,-179.023,9.342,149.564
C04368=1110.437,198.089,-66.776,-179.020,9.345,149.564
C04369=1110.432,198.338,-66.801,-179.018,9.348,149.564
C04370=1110.427,198.587,-66.827,-179.015,9.351,149.564
C04371=1110.424,198.835,-66.852,-179.012,9.354,149.564
C04372=1110.419,199.084,-66.877,-179.010,9.357,149.564
C04373=1110.414,199.333,-66.902,-179.007,9.360,149.564
C04374=1110.409,199.581,-66.927,-179.004,9.363,149.564
C04375=1110.406,199.830,-66.952,-179.002,9.366,149.564
C04376=1110.402,200.043,-66.973,-179.000,9.368,149.564
C04377=1110.398,200.256,-66.995,-178.997,9.371,149.564
C04378=1110.394,200.470,-67.017,-178.995,9.373,149.564
C04379=1110.390,200.682,-67.038,-178.992,9.377,149.564
C04380=1110.387,200.896,-67.060,-178.990,9.379,149.564
C04381=1110.383,201.109,-67.082,-178.988,9.381,149.564
C04382=1110.379,201.321,-67.103,-178.985,9.384,149.564
C04383=1110.375,201.535,-67.125,-178.983,9.386,149.564
C04384=1110.370,201.784,-67.150,-178.980,9.389,149.564
C04385=1110.366,202.032,-67.176,-178.978,9.392,149.564
C04386=1110.362,202.282,-67.201,-178.975,9.395,149.564
C04387=1110.357,202.530,-67.227,-178.972,9.397,149.563
C04388=1110.353,202.778,-67.252,-178.969,9.400,149.563
C04389=1110.348,203.027,-67.276,-178.966,9.403,149.563
C04390=1110.344,203.276,-67.302,-178.963,9.406,149.563
C04391=1110.340,203.525,-67.328,-178.961,9.409,149.563
C04392=1110.335,203.773,-67.353,-178.958,9.412,149.563
C04393=1110.331,204.022,-67.379,-178.955,9.414,149.563
C04394=1110.326,204.271,-67.404,-178.952,9.418,149.563
C04395=1110.321,204.519,-67.429,-178.950,9.420,149.563
C04396=1110.317,204.768,-67.455,-178.947,9.423,149.563
C04397=1110.313,205.017,-67.481,-178.944,9.426,149.563
C04398=1110.308,205.265,-67.506,-178.940,9.430,149.563
C04399=1110.304,205.514,-67.532,-178.938,9.432,149.563
C04400=1110.299,205.763,-67.557,-178.935,9.435,149.562
C04401=1110.294,206.011,-67.582,-178.932,9.438,149.562
C04402=1110.290,206.260,-67.608,-178.929,9.441,149.562
C04403=1110.286,206.509,-67.634,-178.926,9.444,149.562
C04404=1110.281,206.757,-67.659,-178.923,9.447,149.562
C04405=1110.277,207.006,-67.685,-178.920,9.449,149.562
C04406=1110.273,207.255,-67.711,-178.918,9.452,149.562
C04407=1110.269,207.503,-67.737,-178.915,9.455,149.562
C04408=1110.264,207.751,-67.762,-178.911,9.459,149.562
C04409=1110.259,208.000,-67.788,-178.908,9.461,149.562
C04410=1110.255,208.249,-67.813,-178.906,9.464,149.562
C04411=1110.251,208.498,-67.839,-178.903,9.467,149.561
C04412=1110.245,208.746,-67.865,-178.900,9.470,149.561
C04413=1110.241,208.995,-67.891,-178.897,9.473,149.561
C04414=1110.237,209.244,-67.917,-178.894,9.477,149.561
C04415=1110.233,209.492,-67.943,-178.891,9.479,149.561
C04416=1110.228,209.740,-67.969,-178.888,9.482,149.561
C04417=1110.224,209.989,-67.994,-178.885,9.485,149.561
C04418=1110.220,210.238,-68.020,-178.882,9.489,149.561
C04419=1110.215,210.487,-68.046,-178.879,9.491,149.561
C04420=1110.211,210.736,-68.072,-178.876,9.495,149.561
C04421=1110.206,210.984,-68.098,-178.873,9.497,149.561
C04422=1110.202,211.232,-68.124,-178.870,9.501,149.561
C04423=1110.198,211.481,-68.150,-178.867,9.504,149.561
C04424=1110.193,211.730,-68.176,-178.865,9.507,149.561
C04425=1110.188,211.979,-68.202,-178.861,9.511,149.561
C04426=1110.185,212.227,-68.228,-178.859,9.514,149.561
C04427=1110.180,212.475,-68.254,-178.856,9.516,149.560
C04428=1110.175,212.724,-68.280,-178.852,9.520,149.561
C04429=1110.171,212.972,-68.307,-178.850,9.523,149.560
C04430=1110.167,213.221,-68.332,-178.846,9.527,149.560
C04431=1110.162,213.470,-68.358,-178.843,9.530,149.560
C04432=1110.158,213.683,-68.380,-178.842,9.532,149.561
C04433=1110.155,213.896,-68.403,-178.840,9.535,149.561
C04434=1110.151,214.109,-68.426,-178.838,9.538,149.561
C04435=1110.147,214.322,-68.448,-178.836,9.540,149.561
C04436=1110.144,214.535,-68.470,-178.834,9.543,149.561
C04437=1110.139,214.748,-68.493,-178.832,9.545,149.561
C04438=1110.136,214.961,-68.516,-178.830,9.548,149.561
C04439=1110.132,215.173,-68.537,-178.828,9.550,149.561
C04440=1110.127,215.422,-68.564,-178.826,9.553,149.561
C04441=1110.123,215.671,-68.590,-178.823,9.556,149.561
C04442=1110.119,215.919,-68.616,-178.822,9.559,149.562
C04443=1110.114,216.168,-68.643,-178.819,9.562,149.562
C04444=1110.110,216.417,-68.669,-178.817,9.565,149.562
C04445=1110.105,216.665,-68.696,-178.814,9.568,149.562
C04446=1110.101,216.914,-68.722,-178.813,9.570,149.562
C04447=1110.097,217.162,-68.748,-178.810,9.574,149.562
C04448=1110.092,217.411,-68.774,-178.808,9.577,149.562
C04449=1110.088,217.660,-68.801,-178.805,9.580,149.562
C04450=1110.084,217.908,-68.827,-178.803,9.583,149.562
C04451=1110.079,218.157,-68.854,-178.801,9.586,149.562
C04452=1110.076,218.405,-68.880,-178.799,9.589,149.563
C04453=1110.071,218.654,-68.906,-178.796,9.592,149.563
C04454=1110.067,218.902,-68.933,-178.794,9.595,149.563
C04455=1110.062,219.151,-68.959,-178.791,9.598,149.563
C04456=1110.058,219.400,-68.986,-178.789,9.602,149.563
C04457=1110.053,219.648,-69.013,-178.787,9.604,149.563
C04458=1110.049,219.897,-69.039,-178.785,9.607,149.563
C04459=1110.044,220.145,-69.066,-178.782,9.610,149.563
C04460=1110.040,220.394,-69.092,-178.780,9.614,149.563
C04461=1110.035,220.643,-69.118,-178.778,9.617,149.564
C04462=1110.031,220.891,-69.145,-178.775,9.620,149.564
C04463=1110.027,221.139,-69.172,-178.773,9.622,149.564
C04464=1110.023,221.388,-69.198,-178.771,9.626,149.564
C04465=1110.018,221.637,-69.225,-178.768,9.629,149.564
C04466=1110.014,221.885,-69.251,-178.766,9.632,149.564
C04467=1110.009,222.133,-69.278,-178.763,9.635,149.564
C04468=1110.005,222.382,-69.305,-178.761,9.638,149.564
C04469=1110.000,222.631,-69.331,-178.758,9.642,149.564
C04470=1109.996,222.879,-69.358,-178.756,9.645,149.564
C04471=1109.992,223.127,-69.385,-178.753,9.648,149.564
C04472=1109.987,223.376,-69.412,-178.751,9.651,149.564
C04473=1109.983,223.624,-69.438,-178.749,9.653,149.565
C04474=1109.978,223.873,-69.464,-178.746,9.656,149.565
C04475=1109.974,224.122,-69.492,-178.744,9.659,149.565
C04476=1109.970,224.371,-69.518,-178.741,9.663,149.565
C04477=1109.966,224.619,-69.545,-178.739,9.666,149.565
C04478=1109.961,224.868,-69.572,-178.736,9.669,149.565
C04479=1109.957,225.116,-69.599,-178.734,9.672,149.565
C04480=1109.952,225.364,-69.626,-178.731,9.675,149.565
C04481=1109.948,225.613,-69.653,-178.728,9.678,149.565
C04482=1109.944,225.861,-69.680,-178.726,9.681,149.565
C04483=1109.939,226.109,-69.707,-178.723,9.684,149.565
C04484=1109.935,226.358,-69.734,-178.721,9.687,149.565
C04485=1109.931,226.607,-69.760,-178.718,9.690,149.565
C04486=1109.927,226.855,-69.788,-178.716,9.693,149.565
C04487=1109.922,227.104,-69.815,-178.713,9.696,149.565
C04488=1109.918,227.317,-69.838,-178.711,9.698,149.565
C04489=1109.914,227.529,-69.860,-178.709,9.701,149.565
C04490=1109.911,227.742,-69.883,-178.706,9.704,149.565
C04491=1109.907,227.955,-69.907,-178.705,9.706,149.565
C04492=1109.903,228.168,-69.930,-178.702,9.708,149.565
C04493=1109.900,228.381,-69.953,-178.700,9.711,149.565
C04494=1109.896,228.594,-69.977,-178.698,9.714,149.565
C04495=1109.892,228.807,-70.000,-178.695,9.716,149.565
C04496=1109.887,229.055,-70.027,-178.692,9.719,149.565
C04497=1109.883,229.304,-70.055,-178.690,9.721,149.565
C04498=1109.879,229.552,-70.081,-178.688,9.724,149.565
C04499=1109.875,229.801,-70.108,-178.685,9.728,149.565
C04500=1109.870,230.049,-70.135,-178.682,9.730,149.565
C04501=1109.866,230.297,-70.163,-178.679,9.733,149.565
C04502=1109.862,230.546,-70.190,-178.677,9.736,149.565
C04503=1109.857,230.795,-70.217,-178.674,9.739,149.565
C04504=1109.853,231.043,-70.244,-178.671,9.742,149.565
C04505=1109.848,231.292,-70.271,-178.668,9.745,149.565
C04506=1109.845,231.540,-70.299,-178.666,9.748,149.565
C04507=1109.840,231.789,-70.326,-178.663,9.751,149.565
C04508=1109.835,232.037,-70.353,-178.660,9.753,149.565
C04509=1109.831,232.285,-70.381,-178.658,9.756,149.565
C04510=1109.827,232.534,-70.408,-178.655,9.758,149.565
C04511=1109.822,232.783,-70.435,-178.652,9.761,149.565
C04512=1109.818,233.031,-70.463,-178.649,9.764,149.564
C04513=1109.813,233.279,-70.490,-178.646,9.767,149.564
C04514=1109.809,233.528,-70.518,-178.644,9.769,149.564
C04515=1109.806,233.776,-70.545,-178.641,9.772,149.564
C04516=1109.801,234.024,-70.572,-178.639,9.775,149.564
C04517=1109.797,234.274,-70.599,-178.636,9.778,149.564
C04518=1109.793,234.521,-70.627,-178.633,9.780,149.564
C04519=1109.788,234.770,-70.654,-178.630,9.782,149.564
C04520=1109.784,235.019,-70.682,-178.628,9.786,149.564
C04521=1109.780,235.267,-70.709,-178.625,9.788,149.564
C04522=1109.775,235.515,-70.737,-178.623,9.790,149.564
C04523=1109.771,235.764,-70.765,-178.620,9.793,149.564
C04524=1109.767,236.012,-70.792,-178.617,9.796,149.563
C04525=1109.762,236.260,-70.819,-178.614,9.799,149.564
C04526=1109.758,236.509,-70.848,-178.612,9.801,149.563
C04527=1109.753,236.758,-70.875,-178.609,9.804,149.563
C04528=1109.749,237.006,-70.903,-178.606,9.806,149.563
C04529=1109.745,237.255,-70.930,-178.604,9.808,149.563
C04530=1109.740,237.503,-70.958,-178.601,9.811,149.563
C04531=1109.736,237.751,-70.985,-178.598,9.814,149.563
C04532=1109.732,238.000,-71.013,-178.595,9.817,149.563
C04533=1109.727,238.248,-71.041,-178.593,9.819,149.563
C04534=1109.723,238.497,-71.069,-178.591,9.822,149.563
C04535=1109.719,238.745,-71.096,-178.588,9.825,149.563
C04536=1109.714,238.993,-71.125,-178.585,9.827,149.563
C04537=1109.710,239.242,-71.152,-178.582,9.829,149.562
C04538=1109.706,239.490,-71.180,-178.580,9.833,149.562
C04539=1109.702,239.739,-71.208,-178.577,9.835,149.562
C04540=1109.697,239.987,-71.235,-178.575,9.837,149.562
C04541=1109.693,240.235,-71.263,-178.572,9.839,149.562
C04542=1109.688,240.484,-71.292,-178.570,9.842,149.562
C04543=1109.684,240.732,-71.319,-178.567,9.845,149.562
C04544=1109.680,240.945,-71.343,-178.564,9.847,149.562
C04545=1109.676,241.158,-71.366,-178.563,9.849,149.562
C04546=1109.673,241.370,-71.391,-178.560,9.851,149.562
C04547=1109.669,241.583,-71.414,-178.558,9.854,149.562
C04548=1109.666,241.796,-71.438,-178.556,9.856,149.562
C04549=1109.662,242.009,-71.462,-178.554,9.858,149.562
C04550=1109.658,242.221,-71.487,-178.551,9.861,149.562
C04551=1109.654,242.434,-71.510,-178.549,9.863,149.562
C04552=1109.651,242.683,-71.538,-178.547,9.865,149.562
C04553=1109.646,242.931,-71.566,-178.544,9.868,149.561
C04554=1109.642,243.179,-71.594,-178.542,9.871,149.562
C04555=1109.637,243.428,-71.623,-178.539,9.873,149.561
C04556=1109.633,243.677,-71.650,-178.537,9.876,149.562
C04557=1109.629,243.925,-71.678,-178.534,9.879,149.561
C04558=1109.624,244.174,-71.707,-178.532,9.881,149.561
C04559=1109.620,244.421,-71.734,-178.529,9.884,149.561
C04560=1109.616,244.670,-71.763,-178.527,9.886,149.561
C04561=1109.611,244.918,-71.791,-178.524,9.889,149.561
C04562=1109.608,245.167,-71.819,-178.522,9.892,149.561
C04563=1109.603,245.415,-71.847,-178.520,9.894,149.561
C04564=1109.599,245.664,-71.876,-178.517,9.897,149.561
C04565=1109.594,245.911,-71.903,-178.514,9.900,149.561
C04566=1109.591,246.160,-71.932,-178.512,9.903,149.561
C04567=1109.585,246.408,-71.960,-178.509,9.905,149.561
C04568=1109.582,246.657,-71.988,-178.507,9.909,149.561
C04569=1109.578,246.905,-72.016,-178.505,9.911,149.561
C04570=1109.573,247.154,-72.045,-178.502,9.914,149.562
C04571=1109.569,247.402,-72.073,-178.500,9.917,149.562
C04572=1109.564,247.650,-72.101,-178.497,9.920,149.562
C04573=1109.560,247.899,-72.129,-178.494,9.923,149.562
C04574=1109.555,248.147,-72.158,-178.491,9.926,149.562
C04575=1109.552,248.395,-72.186,-178.488,9.929,149.561
C04576=1109.548,248.644,-72.215,-178.485,9.932,149.561
C04577=1109.543,248.892,-72.243,-178.481,9.936,149.561
C04578=1109.539,249.140,-72.271,-178.478,9.938,149.561
C04579=1109.534,249.389,-72.299,-178.475,9.941,149.561
C04580=1109.530,249.637,-72.328,-178.472,9.943,149.561
C04581=1109.526,249.885,-72.357,-178.469,9.946,149.561
C04582=1109.522,250.133,-72.385,-178.466,9.949,149.560
C04583=1109.517,250.382,-72.414,-178.463,9.952,149.560
C04584=1109.514,250.631,-72.442,-178.460,9.954,149.560
C04585=1109.509,250.878,-72.471,-178.457,9.957,149.560
C04586=1109.505,251.127,-72.499,-178.454,9.960,149.560
C04587=1109.501,251.376,-72.528,-178.451,9.962,149.560
C04588=1109.496,251.624,-72.555,-178.448,9.965,149.560
C04589=1109.492,251.872,-72.585,-178.445,9.967,149.559
C04590=1109.488,252.121,-72.614,-178.443,9.969,149.559
C04591=1109.483,252.369,-72.641,-178.440,9.972,149.559
C04592=1109.479,252.617,-72.671,-178.437,9.974,149.559
C04593=1109.475,252.866,-72.699,-178.434,9.977,149.559
C04594=1109.470,253.113,-72.728,-178.431,9.979,149.558
C04595=1109.466,253.362,-72.757,-178.429,9.981,149.558
C04596=1109.462,253.611,-72.785,-178.426,9.984,149.558
C04597=1109.457,253.858,-72.814,-178.423,9.986,149.558
C04598=1109.453,254.107,-72.843,-178.420,9.989,149.558
C04599=1109.450,254.355,-72.872,-178.418,9.991,149.558
C04600=1109.445,254.568,-72.896,-178.416,9.993,149.558
C04601=1109.442,254.780,-72.921,-178.414,9.995,149.558
C04602=1109.438,254.993,-72.946,-178.412,9.997,149.558
C04603=1109.435,255.206,-72.970,-178.409,9.999,149.558
C04604=1109.431,255.419,-72.995,-178.407,10.001,149.558
C04605=1109.427,255.631,-73.019,-178.405,10.003,149.557
C04606=1109.423,255.844,-73.044,-178.403,10.006,149.558
C04607=1109.420,256.056,-73.068,-178.401,10.008,149.558
C04608=1109.416,256.304,-73.098,-178.399,10.010,149.557
C04609=1109.411,256.553,-73.127,-178.396,10.013,149.557
C04610=1109.408,256.801,-73.155,-178.394,10.016,149.557
C04611=1109.403,257.049,-73.185,-178.391,10.019,149.557
C04612=1109.398,257.298,-73.213,-178.388,10.021,149.557
C04613=1109.394,257.546,-73.243,-178.385,10.024,149.557
C04614=1109.391,257.794,-73.271,-178.383,10.027,149.557
C04615=1109.386,258.043,-73.300,-178.380,10.029,149.557
C04616=1109.381,258.290,-73.329,-178.377,10.032,149.557
C04617=1109.377,258.539,-73.358,-178.374,10.035,149.557
C04618=1109.374,258.787,-73.387,-178.372,10.038,149.557
C04619=1109.369,259.035,-73.416,-178.369,10.041,149.557
C04620=1109.365,259.284,-73.446,-178.366,10.043,149.557
C04621=1109.361,259.533,-73.474,-178.363,10.046,149.557
C04622=1109.356,259.780,-73.504,-178.360,10.049,149.557
C04623=1109.352,260.028,-73.532,-178.357,10.051,149.556
C04624=1109.348,260.277,-73.561,-178.355,10.054,149.556
C04625=1109.344,260.525,-73.591,-178.352,10.057,149.556
C04626=1109.340,260.774,-73.620,-178.349,10.060,149.556
C04627=1109.335,261.022,-73.649,-178.346,10.062,149.556
C04628=1109.331,261.270,-73.679,-178.343,10.065,149.556
C04629=1109.326,261.518,-73.707,-178.340,10.068,149.556
C04630=1109.322,261.767,-73.737,-178.337,10.071,149.556
C04631=1109.319,262.014,-73.766,-178.334,10.073,149.556
C04632=1109.314,262.263,-73.795,-178.332,10.075,149.556
C04633=1109.310,262.511,-73.825,-178.329,10.078,149.556
C04634=1109.306,262.759,-73.854,-178.326,10.081,149.555
C04635=1109.302,263.008,-73.883,-178.323,10.084,149.555
C04636=1109.297,263.256,-73.912,-178.320,10.086,149.555
C04637=1109.293,263.504,-73.941,-178.317,10.089,149.555
C04638=1109.288,263.752,-73.971,-178.314,10.092,149.555
C04639=1109.284,264.001,-74.000,-178.311,10.095,149.555
C04640=1109.280,264.249,-74.030,-178.308,10.097,149.555
C04641=1109.276,264.497,-74.059,-178.306,10.099,149.554
C04642=1109.272,264.745,-74.089,-178.303,10.102,149.554
C04643=1109.267,264.994,-74.118,-178.300,10.105,149.554
C04644=1109.263,265.242,-74.147,-178.297,10.107,149.554
C04645=1109.259,265.490,-74.177,-178.295,10.109,149.554
C04646=1109.255,265.738,-74.206,-178.292,10.112,149.554
C04647=1109.251,265.987,-74.236,-178.289,10.115,149.554
C04648=1109.247,266.235,-74.265,-178.285,10.117,149.554
C04649=1109.243,266.483,-74.295,-178.283,10.119,149.553
C04650=1109.239,266.731,-74.325,-178.280,10.122,149.553
C04651=1109.234,266.979,-74.355,-178.277,10.125,149.553
C04652=1109.229,267.228,-74.384,-178.274,10.127,149.553
C04653=1109.225,267.476,-74.414,-178.272,10.129,149.553
C04654=1109.221,267.724,-74.443,-178.269,10.132,149.553
C04655=1109.217,267.973,-74.473,-178.266,10.135,149.553
C04656=1109.213,268.185,-74.498,-178.264,10.137,149.553
C04657=1109.209,268.397,-74.524,-178.262,10.139,149.553
C04658=1109.206,268.609,-74.550,-178.259,10.142,149.552
C04659=1109.202,268.822,-74.574,-178.256,10.144,149.552
C04660=1109.199,269.035,-74.600,-178.254,10.146,149.552
C04661=1109.195,269.247,-74.625,-178.252,10.148,149.552
C04662=1109.191,269.459,-74.651,-178.249,10.151,149.552
C04663=1109.188,269.672,-74.676,-178.247,10.153,149.552
C04664=1109.184,269.920,-74.706,-178.244,10.155,149.552
C04665=1109.180,270.168,-74.736,-178.241,10.158,149.552
C04666=1109.175,270.417,-74.766,-178.239,10.160,149.552
C04667=1109.171,270.665,-74.795,-178.236,10.163,149.552
C04668=1109.167,270.913,-74.825,-178.233,10.166,149.552
C04669=1109.163,271.161,-74.855,-178.230,10.169,149.551
C04670=1109.159,271.409,-74.884,-178.227,10.171,149.551
C04671=1109.154,271.657,-74.915,-178.224,10.174,149.551
C04672=1109.150,271.905,-74.944,-178.221,10.176,149.551
C04673=1109.146,272.154,-74.975,-178.218,10.178,149.551
C04674=1109.142,272.402,-75.004,-178.215,10.181,149.551
C04675=1109.137,272.651,-75.034,-178.212,10.184,149.551
C04676=1109.133,272.898,-75.065,-178.210,10.187,149.551
C04677=1109.129,273.146,-75.094,-178.207,10.189,149.550
C04678=1109.125,273.394,-75.124,-178.204,10.191,149.550
C04679=1109.121,273.643,-75.154,-178.201,10.194,149.550
C04680=1109.117,273.890,-75.184,-178.198,10.197,149.550
C04681=1109.113,274.139,-75.214,-178.195,10.200,149.550
C04682=1109.108,274.387,-75.245,-178.193,10.203,149.550
C04683=1109.104,274.636,-75.275,-178.190,10.205,149.550
C04684=1109.100,274.883,-75.305,-178.186,10.208,149.550
C04685=1109.095,275.132,-75.335,-178.184,10.210,149.549
C04686=1109.092,275.379,-75.365,-178.181,10.212,149.549
C04687=1109.088,275.627,-75.395,-178.178,10.215,149.549
C04688=1109.083,275.876,-75.426,-178.175,10.218,149.549
C04689=1109.080,276.124,-75.456,-178.172,10.221,149.549
C04690=1109.075,276.373,-75.486,-178.169,10.224,149.549
C04691=1109.071,276.620,-75.516,-178.166,10.226,149.549
C04692=1109.067,276.868,-75.546,-178.164,10.228,149.549
C04693=1109.063,277.117,-75.576,-178.161,10.231,149.548
C04694=1109.059,277.365,-75.607,-178.158,10.233,149.548
C04695=1109.054,277.613,-75.637,-178.155,10.236,149.548
C04696=1109.050,277.861,-75.667,-178.152,10.239,149.548
C04697=1109.047,278.109,-75.697,-178.149,10.241,149.548
C04698=1109.042,278.357,-75.728,-178.146,10.244,149.548
C04699=1109.038,278.605,-75.758,-178.143,10.247,149.548
C04700=1109.033,278.854,-75.788,-178.140,10.249,149.548
C04701=1109.029,279.101,-75.819,-178.137,10.251,149.547
C04702=1109.025,279.350,-75.850,-178.134,10.254,149.547
C04703=1109.021,279.598,-75.880,-178.131,10.257,149.547
C04704=1109.016,279.846,-75.910,-178.128,10.260,149.547
C04705=1109.013,280.094,-75.940,-178.125,10.262,149.547
C04706=1109.009,280.342,-75.971,-178.122,10.265,149.547
C04707=1109.004,280.590,-76.002,-178.119,10.268,149.547
C04708=1109.000,280.838,-76.032,-178.116,10.269,149.546
C04709=1108.996,281.087,-76.063,-178.113,10.272,149.546
C04710=1108.992,281.334,-76.093,-178.110,10.274,149.546
C04711=1108.987,281.583,-76.123,-178.107,10.277,149.546
C04712=1108.984,281.795,-76.150,-178.105,10.279,149.546
C04713=1108.981,282.007,-76.176,-178.102,10.282,149.546
C04714=1108.977,282.220,-76.203,-178.099,10.284,149.545
C04715=1108.974,282.432,-76.229,-178.097,10.285,149.545
C04716=1108.970,282.644,-76.254,-178.094,10.288,149.545
C04717=1108.967,282.857,-76.281,-178.092,10.290,149.545
C04718=1108.962,283.069,-76.307,-178.089,10.292,149.545
C04719=1108.959,283.281,-76.334,-178.086,10.295,149.545
C04720=1108.955,283.529,-76.364,-178.084,10.297,149.544
C04721=1108.951,283.778,-76.395,-178.081,10.299,149.544
C04722=1108.947,284.025,-76.426,-178.077,10.302,149.544
C04723=1108.942,284.273,-76.456,-178.074,10.305,149.544
C04724=1108.939,284.522,-76.487,-178.071,10.307,149.544
C04725=1108.934,284.770,-76.518,-178.068,10.310,149.544
C04726=1108.930,285.018,-76.548,-178.065,10.313,149.544
C04727=1108.926,285.266,-76.580,-178.062,10.315,149.543
C04728=1108.922,285.514,-76.610,-178.060,10.317,149.543
C04729=1108.918,285.763,-76.641,-178.056,10.319,149.543
C04730=1108.913,286.010,-76.672,-178.053,10.322,149.543
C04731=1108.910,286.258,-76.703,-178.050,10.325,149.542
C04732=1108.905,286.506,-76.734,-178.047,10.327,149.542
C04733=1108.901,286.754,-76.764,-178.044,10.330,149.542
C04734=1108.897,287.003,-76.796,-178.041,10.332,149.542
C04735=1108.893,287.250,-76.827,-178.038,10.335,149.542
C04736=1108.889,287.498,-76.857,-178.035,10.337,149.542
C04737=1108.885,287.747,-76.888,-178.032,10.340,149.542
C04738=1108.880,287.995,-76.919,-178.029,10.342,149.541
C04739=1108.876,288.243,-76.951,-178.026,10.345,149.541
C04740=1108.872,288.491,-76.982,-178.023,10.348,149.541
C04741=1108.868,288.739,-77.012,-178.020,10.350,149.541
C04742=1108.864,288.986,-77.044,-178.017,10.353,149.541
C04743=1108.860,289.235,-77.075,-178.013,10.355,149.540
C04744=1108.856,289.483,-77.106,-178.010,10.358,149.540
C04745=1108.852,289.731,-77.137,-178.008,10.360,149.540
C04746=1108.847,289.979,-77.168,-178.005,10.362,149.540
C04747=1108.843,290.226,-77.198,-178.001,10.365,149.540
C04748=1108.840,290.475,-77.230,-177.999,10.368,149.540
C04749=1108.835,290.722,-77.261,-177.996,10.370,149.540
C04750=1108.831,290.971,-77.293,-177.992,10.373,149.539
C04751=1108.827,291.218,-77.324,-177.989,10.376,149.539
C04752=1108.823,291.467,-77.355,-177.986,10.378,149.539
C04753=1108.819,291.715,-77.387,-177.984,10.380,149.539
C04754=1108.814,291.963,-77.417,-177.980,10.382,149.539
C04755=1108.811,292.211,-77.449,-177.977,10.385,149.538
C04756=1108.806,292.459,-77.480,-177.974,10.388,149.538
C04757=1108.802,292.707,-77.512,-177.971,10.390,149.538
C04758=1108.798,292.955,-77.543,-177.968,10.393,149.538
C04759=1108.794,293.203,-77.574,-177.965,10.396,149.538
C04760=1108.790,293.451,-77.606,-177.962,10.398,149.538
C04761=1108.786,293.699,-77.637,-177.959,10.401,149.537
C04762=1108.781,293.947,-77.669,-177.956,10.403,149.537
C04763=1108.777,294.195,-77.700,-177.953,10.405,149.537
C04764=1108.774,294.443,-77.732,-177.950,10.408,149.537
C04765=1108.769,294.691,-77.763,-177.947,10.410,149.537
C04766=1108.765,294.939,-77.794,-177.944,10.413,149.537
C04767=1108.761,295.187,-77.826,-177.940,10.416,149.536
C04768=1108.758,295.399,-77.852,-177.938,10.418,149.536
C04769=1108.754,295.611,-77.879,-177.936,10.420,149.536
C04770=1108.751,295.824,-77.907,-177.933,10.422,149.536
C04771=1108.748,296.036,-77.933,-177.930,10.424,149.536
C04772=1108.744,296.248,-77.960,-177.928,10.426,149.536
C04773=1108.740,296.460,-77.987,-177.925,10.429,149.535
C04774=1108.737,296.672,-78.015,-177.923,10.431,149.535
C04775=1108.733,296.884,-78.042,-177.920,10.432,149.535
C04776=1108.729,297.133,-78.073,-177.917,10.435,149.535
C04777=1108.725,297.380,-78.104,-177.914,10.438,149.535
C04778=1108.721,297.628,-78.136,-177.911,10.440,149.535
C04779=1108.717,297.876,-78.169,-177.907,10.443,149.534
C04780=1108.713,298.124,-78.200,-177.904,10.446,149.534
C04781=1108.709,298.372,-78.232,-177.901,10.448,149.534
C04782=1108.705,298.621,-78.263,-177.898,10.451,149.534
C04783=1108.701,298.868,-78.295,-177.896,10.452,149.534
C04784=1108.697,299.116,-78.326,-177.893,10.455,149.534
C04785=1108.693,299.364,-78.359,-177.889,10.458,149.533
C04786=1108.688,299.612,-78.390,-177.886,10.460,149.533
C04787=1108.684,299.860,-78.422,-177.883,10.463,149.533
C04788=1108.681,300.108,-78.454,-177.880,10.466,149.533
C04789=1108.676,300.355,-78.486,-177.877,10.468,149.533
C04790=1108.672,300.603,-78.518,-177.874,10.471,149.533
C04791=1108.668,300.851,-78.550,-177.871,10.474,149.532
C04792=1108.665,301.099,-78.582,-177.868,10.475,149.532
C04793=1108.660,301.347,-78.614,-177.865,10.478,149.532
C04794=1108.656,301.595,-78.646,-177.862,10.480,149.532
C04795=1108.652,301.843,-78.677,-177.859,10.483,149.532
C04796=1108.647,302.091,-78.710,-177.856,10.486,149.531
C04797=1108.643,302.339,-78.741,-177.853,10.488,149.531
C04798=1108.640,302.587,-78.773,-177.849,10.491,149.531
C04799=1108.635,302.835,-78.806,-177.846,10.494,149.531
C04800=1108.631,303.083,-78.837,-177.843,10.496,149.531
C04801=1108.627,303.331,-78.869,-177.841,10.498,149.531
C04802=1108.623,303.579,-78.901,-177.837,10.500,149.530
C04803=1108.619,303.826,-78.934,-177.834,10.503,149.530
C04804=1108.614,304.074,-78.966,-177.831,10.506,149.530
C04805=1108.611,304.322,-78.998,-177.828,10.508,149.530
C04806=1108.607,304.570,-79.030,-177.825,10.511,149.530
C04807=1108.603,304.818,-79.062,-177.822,10.513,149.530
C04808=1108.598,305.066,-79.094,-177.819,10.516,149.529
C04809=1108.594,305.314,-79.127,-177.815,10.518,149.529
C04810=1108.590,305.562,-79.159,-177.813,10.520,149.529
C04811=1108.587,305.810,-79.191,-177.810,10.523,149.529
C04812=1108.582,306.058,-79.223,-177.807,10.526,149.529
C04813=1108.579,306.305,-79.256,-177.803,10.528,149.528
C04814=1108.574,306.553,-79.288,-177.801,10.531,149.528
C04815=1108.570,306.801,-79.319,-177.797,10.533,149.528
C04816=1108.566,307.049,-79.353,-177.794,10.536,149.528
C04817=1108.562,307.297,-79.384,-177.791,10.539,149.528
C04818=1108.558,307.545,-79.417,-177.788,10.541,149.528
C04819=1108.554,307.793,-79.449,-177.785,10.543,149.527
C04820=1108.549,308.040,-79.482,-177.782,10.546,149.527
C04821=1108.546,308.288,-79.514,-177.779,10.548,149.527
C04822=1108.541,308.536,-79.547,-177.776,10.551,149.527
C04823=1108.538,308.784,-79.578,-177.773,10.553,149.527
C04824=1108.532,309.089,-79.619,-177.769,10.557,149.527
C04825=1108.527,309.396,-79.659,-177.765,10.560,149.526
C04826=1108.522,309.701,-79.699,-177.762,10.562,149.526
C04827=1108.518,310.008,-79.739,-177.758,10.565,149.526
C04828=1108.514,310.255,-79.772,-177.755,10.568,149.526
C04829=1108.509,310.503,-79.804,-177.751,10.571,149.525
C04830=1108.505,310.751,-79.837,-177.748,10.573,149.525
C04831=1108.501,310.999,-79.869,-177.745,10.576,149.525
C04832=1108.497,311.246,-79.902,-177.742,10.579,149.525
C04833=1108.494,311.494,-79.935,-177.739,10.581,149.525
C04834=1108.489,311.742,-79.967,-177.736,10.583,149.525
C04835=1108.485,311.990,-80.000,-177.733,10.586,149.524
C04836=1108.482,312.238,-80.032,-177.730,10.588,149.524
C04837=1108.477,312.486,-80.065,-177.727,10.591,149.524
C04838=1108.473,312.733,-80.098,-177.724,10.593,149.524
C04839=1108.470,312.981,-80.130,-177.721,10.596,149.524
C04840=1108.465,313.229,-80.163,-177.717,10.598,149.524
C04841=1108.461,313.477,-80.197,-177.714,10.601,149.523
C04842=1108.457,313.725,-80.229,-177.711,10.604,149.523
C04843=1108.453,313.973,-80.262,-177.708,10.605,149.523
C04844=1108.449,314.220,-80.295,-177.706,10.608,149.523
C04845=1108.445,314.468,-80.328,-177.702,10.610,149.523
C04846=1108.441,314.716,-80.360,-177.699,10.613,149.523
C04847=1108.437,314.964,-80.393,-177.696,10.616,149.522
C04848=1108.433,315.212,-80.426,-177.693,10.618,149.522
C04849=1108.429,315.459,-80.459,-177.690,10.621,149.522
C04850=1108.426,315.707,-80.492,-177.686,10.623,149.522
C04851=1108.421,315.955,-80.524,-177.683,10.626,149.522
C04852=1108.417,316.203,-80.557,-177.680,10.629,149.521
C04853=1108.413,316.451,-80.590,-177.678,10.631,149.521
C04854=1108.409,316.698,-80.624,-177.674,10.633,149.521
C04855=1108.405,316.946,-80.656,-177.671,10.635,149.521
C04856=1108.401,317.193,-80.689,-177.668,10.638,149.521
C04857=1108.397,317.441,-80.723,-177.665,10.641,149.521
C04858=1108.394,317.690,-80.756,-177.662,10.643,149.520
C04859=1108.389,317.937,-80.789,-177.659,10.646,149.520
C04860=1108.385,318.185,-80.822,-177.655,10.648,149.520
C04861=1108.382,318.432,-80.855,-177.652,10.651,149.520
C04862=1108.378,318.680,-80.888,-177.650,10.653,149.520
C04863=1108.374,318.928,-80.921,-177.647,10.656,149.520
C04864=1108.369,319.176,-80.954,-177.643,10.658,149.519
C04865=1108.365,319.423,-80.988,-177.640,10.660,149.519
C04866=1108.361,319.671,-81.021,-177.637,10.663,149.519
C04867=1108.357,319.919,-81.054,-177.634,10.666,149.519
C04868=1108.354,320.167,-81.087,-177.631,10.668,149.519
C04869=1108.349,320.415,-81.121,-177.628,10.671,149.518
C04870=1108.345,320.663,-81.154,-177.624,10.673,149.518
C04871=1108.341,320.910,-81.187,-177.622,10.675,149.518
C04872=1108.096,310.158,-79.818,-177.755,10.568,149.526
C04873=1108.101,309.815,-79.773,-177.759,10.564,149.526
C04874=1108.107,309.472,-79.728,-177.763,10.561,149.526
C04875=1108.112,309.129,-79.684,-177.768,10.557,149.526
C04876=1108.118,308.785,-79.638,-177.772,10.554,149.527
C04877=1108.121,308.537,-79.605,-177.775,10.551,149.527
C04878=1108.126,308.290,-79.573,-177.778,10.549,149.527
C04879=1108.130,308.042,-79.541,-177.781,10.546,149.527
C04880=1108.134,307.794,-79.508,-177.784,10.543,149.527
C04881=1108.138,307.546,-79.477,-177.787,10.542,149.528
C04882=1108.142,307.298,-79.443,-177.790,10.539,149.528
C04883=1108.146,307.050,-79.412,-177.793,10.537,149.528
C04884=1108.150,306.802,-79.379,-177.797,10.534,149.528
C04885=1108.154,306.555,-79.347,-177.800,10.531,149.528
C04886=1108.159,306.307,-79.314,-177.803,10.529,149.528
C04887=1108.162,306.059,-79.283,-177.806,10.526,149.529
C04888=1108.166,305.811,-79.250,-177.809,10.524,149.529
C04889=1108.170,305.563,-79.218,-177.812,10.521,149.529
C04890=1108.175,305.316,-79.186,-177.815,10.519,149.529
C04891=1108.179,305.067,-79.154,-177.818,10.516,149.529
C04892=1108.182,304.820,-79.121,-177.821,10.514,149.530
C04893=1108.187,304.572,-79.089,-177.824,10.511,149.530
C04894=1108.191,304.324,-79.057,-177.827,10.509,149.530
C04895=1108.195,304.076,-79.025,-177.830,10.506,149.530
C04896=1108.199,303.828,-78.993,-177.834,10.504,149.530
C04897=1108.203,303.580,-78.960,-177.836,10.501,149.530
C04898=1108.207,303.332,-78.928,-177.840,10.498,149.531
C04899=1108.212,303.085,-78.896,-177.842,10.496,149.531
C04900=1108.215,302.837,-78.865,-177.845,10.494,149.531
C04901=1108.220,302.588,-78.832,-177.848,10.491,149.531
C04902=1108.223,302.340,-78.800,-177.852,10.489,149.531
C04903=1108.228,302.093,-78.769,-177.855,10.486,149.531
C04904=1108.232,301.845,-78.736,-177.858,10.484,149.532
C04905=1108.236,301.597,-78.705,-177.861,10.481,149.532
C04906=1108.240,301.349,-78.673,-177.864,10.478,149.532
C04907=1108.245,301.101,-78.641,-177.867,10.476,149.532
C04908=1108.248,300.853,-78.609,-177.870,10.474,149.532
C04909=1108.252,300.605,-78.577,-177.873,10.471,149.532
C04910=1108.256,300.357,-78.545,-177.876,10.469,149.533
C04911=1108.261,300.109,-78.513,-177.879,10.466,149.533
C04912=1108.264,299.861,-78.481,-177.882,10.464,149.533
C04913=1108.269,299.614,-78.450,-177.885,10.461,149.533
C04914=1108.272,299.366,-78.418,-177.889,10.458,149.533
C04915=1108.277,299.117,-78.385,-177.892,10.456,149.533
C04916=1108.281,298.870,-78.354,-177.895,10.453,149.534
C04917=1108.285,298.622,-78.322,-177.897,10.451,149.534
C04918=1108.289,298.373,-78.291,-177.901,10.449,149.534
C04919=1108.293,298.126,-78.259,-177.903,10.446,149.534
C04920=1108.297,297.878,-78.228,-177.907,10.444,149.534
C04921=1108.301,297.630,-78.195,-177.910,10.441,149.534
C04922=1108.306,297.382,-78.164,-177.913,10.438,149.535
C04923=1108.309,297.134,-78.132,-177.916,10.436,149.535
C04924=1108.313,296.886,-78.101,-177.919,10.433,149.535
C04925=1108.318,296.674,-78.074,-177.922,10.431,149.535
C04926=1108.320,296.462,-78.047,-177.924,10.429,149.535
C04927=1108.324,296.250,-78.019,-177.927,10.426,149.535
C04928=1108.328,296.037,-77.992,-177.930,10.425,149.536
C04929=1108.331,295.825,-77.966,-177.932,10.423,149.536
C04930=1108.334,295.613,-77.938,-177.935,10.420,149.536
C04931=1108.339,295.401,-77.911,-177.937,10.418,149.536
C04932=1108.342,295.189,-77.885,-177.940,10.416,149.536
C04933=1108.345,294.941,-77.853,-177.943,10.414,149.536
C04934=1108.350,294.693,-77.822,-177.946,10.411,149.537
C04935=1108.354,294.445,-77.790,-177.949,10.408,149.537
C04936=1108.357,294.197,-77.759,-177.952,10.406,149.537
C04937=1108.362,293.949,-77.728,-177.955,10.403,149.537
C04938=1108.366,293.701,-77.696,-177.958,10.401,149.537
C04939=1108.370,293.453,-77.665,-177.961,10.399,149.537
C04940=1108.374,293.205,-77.633,-177.964,10.396,149.538
C04941=1108.378,292.957,-77.602,-177.967,10.394,149.538
C04942=1108.382,292.709,-77.571,-177.970,10.391,149.538
C04943=1108.386,292.461,-77.539,-177.973,10.388,149.538
C04944=1108.391,292.213,-77.508,-177.976,10.386,149.538
C04945=1108.394,291.965,-77.476,-177.980,10.383,149.539
C04946=1108.399,291.717,-77.446,-177.983,10.380,149.539
C04947=1108.403,291.469,-77.414,-177.985,10.379,149.539
C04948=1108.407,291.221,-77.383,-177.988,10.376,149.539
C04949=1108.411,290.973,-77.351,-177.991,10.373,149.539
C04950=1108.416,290.725,-77.320,-177.995,10.371,149.539
C04951=1108.420,290.476,-77.289,-177.997,10.368,149.539
C04952=1108.424,290.229,-77.258,-178.001,10.366,149.540
C04953=1108.427,289.980,-77.227,-178.004,10.363,149.540
C04954=1108.431,289.733,-77.196,-178.007,10.360,149.540
C04955=1108.435,289.484,-77.165,-178.009,10.358,149.540
C04956=1108.440,289.236,-77.134,-178.013,10.356,149.540
C04957=1108.444,288.988,-77.102,-178.016,10.353,149.541
C04958=1108.448,288.740,-77.071,-178.019,10.350,149.541
C04959=1108.453,288.492,-77.040,-178.022,10.348,149.541
C04960=1108.456,288.245,-77.009,-178.025,10.345,149.541
C04961=1108.461,287.997,-76.978,-178.028,10.343,149.541
C04962=1108.465,287.748,-76.947,-178.031,10.340,149.541
C04963=1108.469,287.500,-76.917,-178.034,10.338,149.542
C04964=1108.473,287.252,-76.885,-178.037,10.336,149.542
C04965=1108.477,287.004,-76.854,-178.040,10.333,149.542
C04966=1108.481,286.756,-76.824,-178.043,10.331,149.542
C04967=1108.485,286.508,-76.793,-178.046,10.328,149.542
C04968=1108.490,286.260,-76.762,-178.049,10.325,149.542
C04969=1108.493,286.012,-76.731,-178.052,10.323,149.543
C04970=1108.498,285.764,-76.700,-178.056,10.320,149.543
C04971=1108.502,285.516,-76.669,-178.059,10.317,149.543
C04972=1108.506,285.268,-76.638,-178.061,10.315,149.543
C04973=1108.510,285.020,-76.608,-178.064,10.313,149.543
C04974=1108.514,284.771,-76.577,-178.067,10.310,149.543
C04975=1108.519,284.523,-76.546,-178.070,10.308,149.544
C04976=1108.523,284.276,-76.516,-178.073,10.305,149.544
C04977=1108.526,284.028,-76.484,-178.076,10.302,149.544
C04978=1108.531,283.780,-76.453,-178.080,10.300,149.544
C04979=1108.535,283.532,-76.423,-178.083,10.297,149.544
C04980=1108.539,283.283,-76.392,-178.085,10.295,149.545
C04981=1108.543,283.071,-76.366,-178.088,10.293,149.545
C04982=1108.546,282.859,-76.339,-178.091,10.291,149.545
C04983=1108.550,282.646,-76.313,-178.093,10.289,149.545
C04984=1108.554,282.434,-76.288,-178.096,10.286,149.545
C04985=1108.556,282.222,-76.261,-178.098,10.284,149.545
C04986=1108.561,282.009,-76.235,-178.101,10.282,149.545
C04987=1108.564,281.797,-76.208,-178.104,10.280,149.545
C04988=1108.567,281.584,-76.182,-178.106,10.278,149.546
C04989=1108.572,281.336,-76.152,-178.109,10.275,149.546
C04990=1108.576,281.089,-76.121,-178.112,10.272,149.546
C04991=1108.580,280.841,-76.091,-178.115,10.270,149.546
C04992=1108.584,280.592,-76.060,-178.118,10.268,149.546
C04993=1108.589,280.344,-76.030,-178.121,10.265,149.546
C04994=1108.593,280.096,-75.999,-178.124,10.262,149.547
C04995=1108.597,279.848,-75.969,-178.127,10.260,149.547
C04996=1108.601,279.600,-75.938,-178.130,10.257,149.547
C04997=1108.605,279.352,-75.908,-178.133,10.254,149.547
C04998=1108.610,279.103,-75.878,-178.136,10.253,149.547
C04999=1108.614,278.856,-75.848,-178.139,10.250,149.547
C05000=1108.618,278.607,-75.817,-178.142,10.247,149.548
C05001=1108.622,278.359,-75.786,-178.145,10.245,149.548
C05002=1108.627,278.111,-75.756,-178.148,10.242,149.548
C05003=1108.630,277.863,-75.726,-178.151,10.239,149.548
C05004=1108.634,277.615,-75.696,-178.154,10.237,149.548
C05005=1108.638,277.367,-75.665,-178.157,10.234,149.548
C05006=1108.642,277.119,-75.635,-178.159,10.232,149.548
C05007=1108.647,276.871,-75.605,-178.162,10.229,149.548
C05008=1108.651,276.623,-75.574,-178.165,10.227,149.549
C05009=1108.655,276.374,-75.544,-178.168,10.224,149.549
C05010=1108.659,276.126,-75.514,-178.171,10.221,149.549
C05011=1108.663,275.878,-75.484,-178.174,10.218,149.549
C05012=1108.668,275.630,-75.454,-178.177,10.216,149.549
C05013=1108.672,275.382,-75.423,-178.179,10.214,149.549
C05014=1108.676,275.134,-75.394,-178.182,10.211,149.549
C05015=1108.680,274.885,-75.363,-178.186,10.208,149.550
C05016=1108.684,274.637,-75.333,-178.189,10.206,149.550
C05017=1108.688,274.389,-75.303,-178.191,10.203,149.550
C05018=1108.693,274.141,-75.273,-178.194,10.200,149.550
C05019=1108.697,273.893,-75.243,-178.197,10.197,149.550
C05020=1108.701,273.645,-75.214,-178.200,10.195,149.550
C05021=1108.705,273.396,-75.182,-178.203,10.193,149.550
C05022=1108.709,273.148,-75.153,-178.206,10.190,149.550
C05023=1108.713,272.900,-75.123,-178.208,10.187,149.550
C05024=1108.717,272.652,-75.093,-178.211,10.184,149.550
C05025=1108.722,272.404,-75.063,-178.214,10.182,149.551
C05026=1108.726,272.156,-75.033,-178.217,10.180,149.551
C05027=1108.730,271.908,-75.004,-178.220,10.177,149.551
C05028=1108.735,271.660,-74.973,-178.223,10.174,149.551
C05029=1108.739,271.411,-74.944,-178.226,10.172,149.551
C05030=1108.743,271.164,-74.913,-178.229,10.169,149.551
C05031=1108.747,270.915,-74.884,-178.232,10.166,149.551
C05032=1108.751,270.666,-74.854,-178.234,10.164,149.551
C05033=1108.756,270.418,-74.824,-178.237,10.161,149.552
C05034=1108.760,270.170,-74.794,-178.240,10.159,149.552
C05035=1108.764,269.922,-74.764,-178.243,10.156,149.552
C05036=1108.768,269.674,-74.735,-178.246,10.153,149.552
C05037=1108.772,269.462,-74.709,-178.248,10.151,149.552
C05038=1108.775,269.249,-74.684,-178.250,10.149,149.552
C05039=1108.779,269.037,-74.658,-178.253,10.146,149.552
C05040=1108.783,268.824,-74.633,-178.256,10.144,149.552
C05041=1108.786,268.611,-74.607,-178.258,10.142,149.552
C05042=1108.789,268.399,-74.582,-178.260,10.140,149.552
C05043=1108.793,268.187,-74.556,-178.263,10.137,149.552
C05044=1108.797,267.974,-74.532,-178.265,10.135,149.553
C05045=1108.801,267.726,-74.501,-178.268,10.133,149.553
C05046=1108.805,267.478,-74.472,-178.270,10.131,149.553
C05047=1108.809,267.230,-74.443,-178.273,10.128,149.553
C05048=1108.814,266.981,-74.413,-178.276,10.125,149.553
C05049=1108.818,266.733,-74.383,-178.279,10.122,149.553
C05050=1108.822,266.485,-74.354,-178.282,10.121,149.553
C05051=1108.827,266.236,-74.324,-178.285,10.118,149.554
C05052=1108.831,265.988,-74.295,-178.288,10.115,149.554
C05053=1108.835,265.740,-74.265,-178.291,10.112,149.554
C05054=1108.839,265.492,-74.235,-178.293,10.110,149.554
C05055=1108.843,265.244,-74.206,-178.296,10.108,149.554
C05056=1108.847,264.996,-74.176,-178.299,10.105,149.554
C05057=1108.851,264.747,-74.147,-178.302,10.102,149.554
C05058=1108.856,264.500,-74.118,-178.304,10.100,149.554
C05059=1108.860,264.252,-74.088,-178.307,10.097,149.554
C05060=1108.864,264.003,-74.059,-178.310,10.095,149.555
C05061=1108.869,263.755,-74.029,-178.313,10.092,149.555
C05062=1108.873,263.506,-74.001,-178.316,10.090,149.555
C05063=1108.877,263.258,-73.971,-178.319,10.087,149.555
C05064=1108.881,263.010,-73.942,-178.322,10.084,149.555
C05065=1108.886,262.761,-73.912,-178.324,10.082,149.555
C05066=1108.890,262.513,-73.883,-178.327,10.079,149.555
C05067=1108.894,262.265,-73.853,-178.330,10.077,149.555
C05068=1108.899,262.017,-73.824,-178.333,10.074,149.556
C05069=1108.903,261.769,-73.795,-178.336,10.071,149.556
C05070=1108.907,261.521,-73.765,-178.339,10.068,149.556
C05071=1108.911,261.272,-73.737,-178.342,10.065,149.556
C05072=1108.915,261.024,-73.708,-178.345,10.063,149.556
C05073=1108.919,260.776,-73.678,-178.347,10.061,149.556
C05074=1108.923,260.527,-73.649,-178.350,10.058,149.556
C05075=1108.928,260.279,-73.619,-178.353,10.055,149.556
C05076=1108.933,260.031,-73.591,-178.356,10.052,149.556
C05077=1108.937,259.783,-73.561,-178.359,10.049,149.556
C05078=1108.940,259.535,-73.533,-178.362,10.047,149.556
C05079=1108.945,259.286,-73.504,-178.365,10.044,149.557
C05080=1108.949,259.038,-73.474,-178.368,10.041,149.557
C05081=1108.953,258.789,-73.445,-178.370,10.039,149.557
C05082=1108.958,258.542,-73.416,-178.372,10.036,149.557
C05083=1108.962,258.293,-73.388,-178.375,10.033,149.557
C05084=1108.966,258.045,-73.358,-178.378,10.030,149.557
C05085=1108.970,257.797,-73.329,-178.381,10.028,149.557
C05086=1108.975,257.548,-73.300,-178.384,10.025,149.557
C05087=1108.979,257.300,-73.272,-178.387,10.022,149.557
C05088=1108.983,257.052,-73.243,-178.389,10.020,149.557
C05089=1108.987,256.803,-73.213,-178.391,10.017,149.557
C05090=1108.992,256.554,-73.185,-178.394,10.014,149.557
C05091=1108.996,256.307,-73.156,-178.397,10.011,149.557
C05092=1109.000,256.059,-73.127,-178.400,10.008,149.557
C05093=1109.004,255.846,-73.102,-178.402,10.006,149.557
C05094=1109.007,255.633,-73.077,-178.404,10.004,149.557
C05095=1109.011,255.420,-73.053,-178.406,10.002,149.557
C05096=1109.015,255.208,-73.028,-178.408,10.000,149.557
C05097=1109.019,254.995,-73.003,-178.411,9.998,149.557
C05098=1109.022,254.783,-72.979,-178.413,9.996,149.558
C05099=1109.026,254.570,-72.954,-178.415,9.993,149.558
C05100=1109.029,254.358,-72.929,-178.417,9.991,149.558
C05101=1109.034,254.109,-72.901,-178.419,9.989,149.558
C05102=1109.038,253.861,-72.873,-178.422,9.986,149.558
C05103=1109.042,253.613,-72.843,-178.425,9.985,149.558
C05104=1109.047,253.364,-72.815,-178.428,9.982,149.558
C05105=1109.050,253.117,-72.786,-178.430,9.980,149.558
C05106=1109.055,252.868,-72.757,-178.433,9.977,149.559
C05107=1109.059,252.619,-72.729,-178.436,9.975,149.559
C05108=1109.063,252.371,-72.700,-178.439,9.973,149.559
C05109=1109.068,252.123,-72.671,-178.441,9.970,149.559
C05110=1109.071,251.875,-72.642,-178.445,9.968,149.559
C05111=1109.076,251.626,-72.614,-178.447,9.966,149.559
C05112=1109.080,251.378,-72.586,-178.450,9.963,149.560
C05113=1109.085,251.129,-72.557,-178.453,9.960,149.560
C05114=1109.089,250.882,-72.529,-178.456,9.958,149.560
C05115=1109.093,250.633,-72.500,-178.459,9.955,149.560
C05116=1109.097,250.384,-72.472,-178.462,9.953,149.560
C05117=1109.102,250.137,-72.443,-178.465,9.950,149.560
C05118=1109.106,249.888,-72.415,-178.468,9.947,149.560
C05119=1109.110,249.639,-72.386,-178.471,9.945,149.561
C05120=1109.114,249.391,-72.358,-178.474,9.942,149.561
C05121=1109.119,249.142,-72.329,-178.477,9.939,149.561
C05122=1109.123,248.895,-72.301,-178.480,9.936,149.561
C05123=1109.127,248.646,-72.272,-178.483,9.933,149.561
C05124=1109.131,248.398,-72.244,-178.486,9.930,149.561
C05125=1109.136,248.150,-72.216,-178.489,9.927,149.561
C05126=1109.140,247.901,-72.187,-178.492,9.924,149.561
C05127=1109.145,247.653,-72.159,-178.495,9.921,149.561
C05128=1109.149,247.404,-72.131,-178.498,9.918,149.561
C05129=1109.153,247.156,-72.103,-178.500,9.915,149.561
C05130=1109.158,246.907,-72.074,-178.503,9.912,149.561
C05131=1109.161,246.659,-72.046,-178.505,9.910,149.561
C05132=1109.166,246.411,-72.018,-178.508,9.907,149.561
C05133=1109.170,246.162,-71.990,-178.510,9.903,149.561
C05134=1109.175,245.914,-71.962,-178.512,9.902,149.561
C05135=1109.179,245.665,-71.933,-178.515,9.898,149.561
C05136=1109.183,245.417,-71.905,-178.518,9.895,149.561
C05137=1109.187,245.169,-71.877,-178.520,9.893,149.561
C05138=1109.192,244.921,-71.849,-178.522,9.890,149.561
C05139=1109.196,244.672,-71.821,-178.525,9.887,149.561
C05140=1109.200,244.424,-71.793,-178.527,9.885,149.561
C05141=1109.205,244.175,-71.764,-178.530,9.882,149.561
C05142=1109.209,243.928,-71.736,-178.533,9.879,149.561
C05143=1109.213,243.679,-71.708,-178.535,9.877,149.561
C05144=1109.218,243.431,-71.680,-178.538,9.874,149.561
C05145=1109.222,243.182,-71.652,-178.540,9.871,149.561
C05146=1109.226,242.934,-71.624,-178.542,9.869,149.561
C05147=1109.230,242.685,-71.597,-178.545,9.866,149.561
C05148=1109.235,242.437,-71.568,-178.548,9.863,149.561
C05149=1109.239,242.225,-71.544,-178.550,9.861,149.562
C05150=1109.242,242.011,-71.521,-178.552,9.859,149.561
C05151=1109.246,241.799,-71.496,-178.554,9.857,149.562
C05152=1109.250,241.586,-71.473,-178.557,9.855,149.562
C05153=1109.253,241.374,-71.449,-178.559,9.853,149.562
C05154=1109.257,241.161,-71.425,-178.561,9.851,149.562
C05155=1109.260,240.948,-71.401,-178.563,9.848,149.562
C05156=1109.265,240.735,-71.377,-178.566,9.846,149.562
C05157=1109.268,240.486,-71.349,-178.568,9.844,149.562
C05158=1109.273,240.238,-71.321,-178.571,9.840,149.562
C05159=1109.277,239.989,-71.293,-178.573,9.838,149.562
C05160=1109.281,239.741,-71.266,-178.576,9.836,149.562
C05161=1109.285,239.494,-71.238,-178.579,9.833,149.562
C05162=1109.290,239.244,-71.210,-178.581,9.830,149.562
C05163=1109.295,238.996,-71.182,-178.584,9.828,149.562
C05164=1109.298,238.748,-71.154,-178.587,9.825,149.562
C05165=1109.303,238.499,-71.127,-178.589,9.822,149.563
C05166=1109.307,238.251,-71.099,-178.591,9.820,149.563
C05167=1109.311,238.003,-71.071,-178.594,9.817,149.563
C05168=1109.316,237.754,-71.044,-178.597,9.815,149.563
C05169=1109.320,237.506,-71.016,-178.600,9.813,149.563
C05170=1109.325,237.257,-70.988,-178.603,9.810,149.563
C05171=1109.329,237.009,-70.960,-178.605,9.807,149.563
C05172=1109.333,236.760,-70.932,-178.607,9.805,149.563
C05173=1109.338,236.512,-70.905,-178.610,9.802,149.563
C05174=1109.342,236.264,-70.877,-178.613,9.799,149.563
C05175=1109.346,236.015,-70.850,-178.616,9.796,149.563
C05176=1109.350,235.767,-70.822,-178.618,9.794,149.563
C05177=1109.355,235.518,-70.795,-178.621,9.791,149.564
C05178=1109.359,235.270,-70.767,-178.624,9.789,149.564
C05179=1109.364,235.021,-70.740,-178.627,9.786,149.564
C05180=1109.368,234.773,-70.712,-178.629,9.784,149.564
C05181=1109.372,234.524,-70.685,-178.632,9.781,149.564
C05182=1109.377,234.276,-70.658,-178.635,9.778,149.564
C05183=1109.381,234.028,-70.630,-178.638,9.775,149.564
C05184=1109.385,233.779,-70.602,-178.640,9.773,149.564
C05185=1109.389,233.531,-70.575,-178.642,9.770,149.564
C05186=1109.394,233.282,-70.548,-178.645,9.768,149.564
C05187=1109.399,233.034,-70.520,-178.648,9.764,149.564
C05188=1109.402,232.785,-70.492,-178.650,9.762,149.564
C05189=1109.407,232.537,-70.465,-178.653,9.760,149.564
C05190=1109.412,232.288,-70.438,-178.656,9.757,149.564
C05191=1109.415,232.040,-70.411,-178.659,9.754,149.565
C05192=1109.419,231.791,-70.384,-178.662,9.751,149.565
C05193=1109.424,231.543,-70.357,-178.664,9.748,149.565
C05194=1109.429,231.294,-70.329,-178.666,9.746,149.565
C05195=1109.432,231.046,-70.301,-178.669,9.743,149.565
C05196=1109.437,230.797,-70.274,-178.672,9.740,149.565
C05197=1109.442,230.549,-70.247,-178.675,9.737,149.565
C05198=1109.446,230.300,-70.220,-178.677,9.734,149.565
C05199=1109.450,230.053,-70.193,-178.680,9.732,149.565
C05200=1109.454,229.804,-70.166,-178.683,9.728,149.565
C05201=1109.459,229.555,-70.138,-178.686,9.726,149.565
C05202=1109.463,229.307,-70.111,-178.688,9.723,149.565
C05203=1109.468,229.058,-70.084,-178.691,9.720,149.565
C05204=1109.472,228.809,-70.057,-178.693,9.717,149.565
C05205=1109.476,228.597,-70.034,-178.696,9.714,149.565
C05206=1109.479,228.384,-70.011,-178.698,9.712,149.565
C05207=1109.483,228.171,-69.987,-178.701,9.709,149.565
C05208=1109.487,227.958,-69.964,-178.702,9.707,149.565
C05209=1109.491,227.746,-69.941,-178.704,9.705,149.565
C05210=1109.494,227.533,-69.918,-178.707,9.702,149.565
C05211=1109.498,227.319,-69.895,-178.709,9.700,149.565
C05212=1109.502,227.106,-69.872,-178.711,9.697,149.565
C05213=1109.506,226.858,-69.845,-178.714,9.694,149.565
C05214=1109.511,226.610,-69.818,-178.716,9.691,149.565
C05215=1109.515,226.361,-69.791,-178.719,9.688,149.565
C05216=1109.519,226.113,-69.764,-178.722,9.685,149.565
C05217=1109.524,225.864,-69.737,-178.724,9.682,149.565
C05218=1109.528,225.616,-69.710,-178.727,9.679,149.565
C05219=1109.532,225.367,-69.683,-178.729,9.676,149.565
C05220=1109.536,225.118,-69.656,-178.732,9.673,149.565
C05221=1109.541,224.870,-69.629,-178.734,9.670,149.565
C05222=1109.545,224.622,-69.603,-178.737,9.666,149.564
C05223=1109.550,224.373,-69.576,-178.739,9.663,149.564
C05224=1109.554,224.125,-69.549,-178.741,9.661,149.564
C05225=1109.558,223.877,-69.522,-178.744,9.658,149.564
C05226=1109.563,223.628,-69.495,-178.746,9.655,149.564
C05227=1109.568,223.379,-69.469,-178.749,9.652,149.564
C05228=1109.572,223.131,-69.442,-178.751,9.649,149.564
C05229=1109.576,222.882,-69.415,-178.754,9.645,149.564
C05230=1109.580,222.633,-69.389,-178.756,9.642,149.564
C05231=1109.584,222.385,-69.361,-178.759,9.639,149.564
C05232=1109.589,222.136,-69.335,-178.761,9.636,149.564
C05233=1109.593,221.888,-69.309,-178.764,9.633,149.564
C05234=1109.598,221.639,-69.282,-178.766,9.631,149.564
C05235=1109.602,221.391,-69.255,-178.768,9.627,149.563
C05236=1109.607,221.142,-69.229,-178.770,9.624,149.563
C05237=1109.611,220.894,-69.202,-178.773,9.621,149.563
C05238=1109.615,220.645,-69.175,-178.775,9.618,149.563
C05239=1109.619,220.397,-69.149,-178.778,9.615,149.563
C05240=1109.624,220.148,-69.122,-178.781,9.612,149.563
C05241=1109.628,219.900,-69.096,-178.782,9.609,149.563
C05242=1109.633,219.651,-69.069,-178.785,9.606,149.563
C05243=1109.637,219.402,-69.043,-178.787,9.603,149.563
C05244=1109.642,219.154,-69.016,-178.790,9.600,149.563
C05245=1109.646,218.906,-68.990,-178.792,9.597,149.563
C05246=1109.651,218.657,-68.963,-178.794,9.593,149.562
C05247=1109.655,218.408,-68.937,-178.796,9.591,149.562
C05248=1109.660,218.159,-68.911,-178.799,9.588,149.562
C05249=1109.663,217.911,-68.884,-178.801,9.584,149.562
C05250=1109.668,217.663,-68.857,-178.804,9.581,149.562
C05251=1109.672,217.414,-68.831,-178.806,9.578,149.562
C05252=1109.676,217.166,-68.805,-178.808,9.576,149.562
C05253=1109.681,216.917,-68.778,-178.810,9.572,149.562
C05254=1109.685,216.668,-68.752,-178.813,9.569,149.562
C05255=1109.689,216.420,-68.726,-178.815,9.566,149.561
C05256=1109.694,216.171,-68.699,-178.817,9.564,149.561
C05257=1109.698,215.922,-68.673,-178.819,9.560,149.561
C05258=1109.703,215.674,-68.647,-178.822,9.557,149.561
C05259=1109.708,215.426,-68.621,-178.824,9.554,149.561
C05260=1109.712,215.177,-68.595,-178.826,9.552,149.561
C05261=1109.716,214.964,-68.572,-178.828,9.548,149.561
C05262=1109.720,214.751,-68.550,-178.830,9.546,149.561
C05263=1109.723,214.538,-68.528,-178.832,9.544,149.561
C05264=1109.727,214.325,-68.504,-178.834,9.541,149.561
C05265=1109.730,214.112,-68.482,-178.835,9.539,149.560
C05266=1109.735,213.899,-68.460,-178.837,9.536,149.560
C05267=1109.738,213.686,-68.438,-178.839,9.534,149.560
C05268=1109.742,213.473,-68.416,-178.842,9.531,149.560
C05269=1109.746,213.224,-68.388,-178.844,9.528,149.560
C05270=1109.751,212.975,-68.363,-178.848,9.524,149.560
C05271=1109.755,212.727,-68.337,-178.850,9.521,149.560
C05272=1109.759,212.479,-68.311,-178.853,9.518,149.560
C05273=1109.764,212.230,-68.285,-178.856,9.515,149.560
C05274=1109.769,211.981,-68.259,-178.859,9.512,149.560
C05275=1109.772,211.733,-68.232,-178.863,9.508,149.560
C05276=1109.777,211.484,-68.207,-178.866,9.505,149.560
C05277=1109.782,211.236,-68.181,-178.868,9.502,149.560
C05278=1109.786,210.987,-68.155,-178.872,9.499,149.560
C05279=1109.791,210.738,-68.129,-178.875,9.496,149.561
C05280=1109.795,210.490,-68.103,-178.877,9.493,149.561
C05281=1109.799,210.241,-68.077,-178.881,9.489,149.561
C05282=1109.803,209.992,-68.051,-178.884,9.486,149.561
C05283=1109.809,209.744,-68.025,-178.886,9.483,149.561
C05284=1109.813,209.495,-67.999,-178.889,9.481,149.561
C05285=1109.817,209.246,-67.974,-178.893,9.477,149.561
C05286=1109.821,208.997,-67.948,-178.895,9.474,149.561
C05287=1109.826,208.750,-67.922,-178.898,9.471,149.561
C05288=1109.830,208.501,-67.896,-178.901,9.468,149.561
C05289=1109.834,208.252,-67.870,-178.904,9.465,149.561
C05290=1109.839,208.004,-67.845,-178.907,9.462,149.561
C05291=1109.844,207.755,-67.819,-178.910,9.459,149.561
C05292=1109.848,207.506,-67.793,-178.913,9.456,149.562
C05293=1109.853,207.258,-67.767,-178.916,9.453,149.562
C05294=1109.857,207.009,-67.741,-178.919,9.450,149.562
C05295=1109.862,206.761,-67.716,-178.922,9.448,149.562
C05296=1109.866,206.512,-67.690,-178.924,9.445,149.562
C05297=1109.870,206.263,-67.664,-178.927,9.442,149.562
C05298=1109.875,206.014,-67.640,-178.931,9.438,149.562
C05299=1109.879,205.765,-67.614,-178.934,9.436,149.562
C05300=1109.884,205.517,-67.588,-178.936,9.433,149.562
C05301=1109.888,205.269,-67.563,-178.939,9.430,149.562
C05302=1109.893,205.020,-67.537,-178.942,9.427,149.562
C05303=1109.897,204.771,-67.511,-178.945,9.424,149.563
C05304=1109.902,204.523,-67.486,-178.948,9.421,149.563
C05305=1109.906,204.274,-67.460,-178.950,9.418,149.563
C05306=1109.910,204.025,-67.435,-178.953,9.416,149.563
C05307=1109.915,203.777,-67.410,-178.956,9.413,149.563
C05308=1109.920,203.528,-67.384,-178.959,9.410,149.563
C05309=1109.924,203.279,-67.358,-178.962,9.407,149.563
C05310=1109.929,203.031,-67.333,-178.965,9.404,149.563
C05311=1109.932,202.782,-67.308,-178.968,9.402,149.563
C05312=1109.937,202.533,-67.283,-178.970,9.398,149.563
C05313=1109.941,202.285,-67.257,-178.973,9.396,149.563
C05314=1109.946,202.035,-67.232,-178.976,9.393,149.563
C05315=1109.951,201.787,-67.207,-178.979,9.390,149.563
C05316=1109.955,201.538,-67.181,-178.982,9.387,149.564
C05317=1109.959,201.325,-67.160,-178.983,9.385,149.564
C05318=1109.962,201.112,-67.138,-178.986,9.382,149.564
C05319=1109.966,200.899,-67.116,-178.988,9.380,149.564
C05320=1109.971,200.686,-67.095,-178.991,9.377,149.564
C05321=1109.974,200.473,-67.073,-178.993,9.375,149.564
C05322=1109.978,200.259,-67.052,-178.995,9.372,149.564
C05323=1109.981,200.047,-67.030,-178.998,9.370,149.564
C05324=1109.985,199.833,-67.009,-179.000,9.367,149.564
C05325=1109.990,199.585,-66.983,-179.002,9.364,149.564
C05326=1109.994,199.336,-66.958,-179.005,9.361,149.564
C05327=1109.999,199.088,-66.933,-179.008,9.358,149.564
C05328=1110.003,198.839,-66.908,-179.010,9.355,149.564
C05329=1110.008,198.590,-66.883,-179.013,9.352,149.564
C05330=1110.012,198.342,-66.857,-179.016,9.349,149.564
C05331=1110.017,198.093,-66.833,-179.018,9.346,149.564
C05332=1110.021,197.844,-66.808,-179.021,9.343,149.564
C05333=1110.026,197.596,-66.783,-179.023,9.340,149.564
C05334=1110.030,197.347,-66.757,-179.026,9.337,149.564
C05335=1110.034,197.097,-66.732,-179.029,9.334,149.564
C05336=1110.039,196.849,-66.708,-179.031,9.331,149.564
C05337=1110.043,196.600,-66.682,-179.034,9.328,149.564
C05338=1110.048,196.351,-66.658,-179.035,9.325,149.564
C05339=1110.052,196.104,-66.633,-179.038,9.322,149.563
C05340=1110.057,195.854,-66.608,-179.040,9.319,149.563
C05341=1110.062,195.605,-66.583,-179.042,9.317,149.563
C05342=1110.065,195.357,-66.558,-179.044,9.313,149.563
C05343=1110.071,195.108,-66.533,-179.046,9.311,149.563
C05344=1110.074,194.860,-66.508,-179.049,9.308,149.563
C05345=1110.079,194.611,-66.484,-179.051,9.305,149.563
C05346=1110.084,194.362,-66.459,-179.053,9.302,149.563
C05347=1110.088,194.113,-66.434,-179.055,9.300,149.563
C05348=1110.092,193.864,-66.409,-179.057,9.296,149.563
C05349=1110.097,193.616,-66.384,-179.059,9.294,149.563
C05350=1110.102,193.367,-66.360,-179.062,9.291,149.563
C05351=1110.106,193.118,-66.334,-179.064,9.288,149.563
C05352=1110.110,192.870,-66.310,-179.066,9.286,149.562
C05353=1110.115,192.621,-66.285,-179.068,9.282,149.562
C05354=1110.119,192.372,-66.261,-179.070,9.280,149.562
C05355=1110.124,192.123,-66.235,-179.073,9.277,149.562
C05356=1110.128,191.875,-66.211,-179.074,9.274,149.562
C05357=1110.133,191.626,-66.187,-179.077,9.271,149.562
C05358=1110.138,191.377,-66.161,-179.079,9.269,149.562
C05359=1110.142,191.128,-66.137,-179.081,9.266,149.562
C05360=1110.147,190.879,-66.112,-179.084,9.263,149.562
C05361=1110.151,190.631,-66.088,-179.086,9.260,149.562
C05362=1110.156,190.383,-66.063,-179.088,9.257,149.562
C05363=1110.160,190.133,-66.038,-179.090,9.255,149.562
C05364=1110.165,189.885,-66.014,-179.093,9.252,149.562
C05365=1110.169,189.636,-65.990,-179.095,9.249,149.562
C05366=1110.174,189.387,-65.965,-179.097,9.246,149.562
C05367=1110.178,189.138,-65.941,-179.100,9.243,149.562
C05368=1110.182,188.890,-65.917,-179.102,9.241,149.562
C05369=1110.187,188.641,-65.892,-179.104,9.238,149.561
C05370=1110.191,188.392,-65.867,-179.107,9.235,149.561
C05371=1110.196,188.143,-65.843,-179.109,9.232,149.561
C05372=1110.200,187.894,-65.818,-179.111,9.229,149.561
C05373=1110.204,187.681,-65.797,-179.113,9.227,149.561
C05374=1110.209,187.468,-65.776,-179.115,9.225,149.561
C05375=1110.212,187.255,-65.756,-179.117,9.222,149.561
C05376=1110.216,187.042,-65.734,-179.119,9.220,149.561
C05377=1110.220,186.829,-65.714,-179.121,9.218,149.561
C05378=1110.224,186.615,-65.693,-179.123,9.214,149.561
C05379=1110.228,186.402,-65.672,-179.125,9.212,149.561
C05380=1110.232,186.189,-65.651,-179.127,9.210,149.561
C05381=1110.236,185.940,-65.626,-179.129,9.207,149.561
C05382=1110.241,185.691,-65.602,-179.131,9.204,149.561
C05383=1110.245,185.443,-65.578,-179.134,9.201,149.561
C05384=1110.250,185.194,-65.553,-179.136,9.198,149.561
C05385=1110.254,184.945,-65.529,-179.138,9.196,149.561
C05386=1110.258,184.697,-65.505,-179.141,9.193,149.561
C05387=1110.263,184.448,-65.481,-179.143,9.190,149.561
C05388=1110.268,184.198,-65.456,-179.145,9.187,149.561
C05389=1110.272,183.950,-65.432,-179.148,9.184,149.561
C05390=1110.276,183.702,-65.408,-179.150,9.181,149.561
C05391=1110.282,183.453,-65.384,-179.153,9.178,149.561
C05392=1110.286,183.203,-65.360,-179.155,9.176,149.561
C05393=1110.290,182.955,-65.336,-179.157,9.172,149.560
C05394=1110.294,182.706,-65.312,-179.160,9.169,149.560
C05395=1110.300,182.457,-65.287,-179.162,9.166,149.560
C05396=1110.304,182.208,-65.264,-179.164,9.164,149.560
C05397=1110.308,181.959,-65.239,-179.167,9.161,149.560
C05398=1110.312,181.711,-65.215,-179.169,9.158,149.560
C05399=1110.318,181.462,-65.191,-179.172,9.155,149.560
C05400=1110.322,181.213,-65.167,-179.174,9.152,149.560
C05401=1110.327,180.965,-65.143,-179.176,9.149,149.560
C05402=1110.330,180.716,-65.119,-179.179,9.146,149.560
C05403=1110.335,180.467,-65.095,-179.181,9.143,149.560
C05404=1110.340,180.218,-65.071,-179.184,9.140,149.560
C05405=1110.345,179.969,-65.047,-179.186,9.136,149.560
C05406=1110.349,179.720,-65.023,-179.188,9.133,149.560
C05407=1110.354,179.472,-64.999,-179.191,9.130,149.560
C05408=1110.358,179.222,-64.975,-179.193,9.128,149.560
C05409=1110.362,178.974,-64.951,-179.195,9.124,149.559
C05410=1110.367,178.725,-64.927,-179.197,9.121,149.559
C05411=1110.371,178.476,-64.904,-179.199,9.119,149.559
C05412=1110.376,178.228,-64.880,-179.201,9.115,149.559
C05413=1110.380,177.979,-64.856,-179.204,9.112,149.559
C05414=1110.386,177.730,-64.832,-179.206,9.110,149.559
C05415=1110.390,177.481,-64.808,-179.208,9.107,149.559
C05416=1110.394,177.232,-64.784,-179.210,9.103,149.559
C05417=1110.399,176.983,-64.761,-179.212,9.101,149.559
C05418=1110.403,176.735,-64.737,-179.215,9.098,149.559
C05419=1110.408,176.486,-64.713,-179.216,9.095,149.558
C05420=1110.412,176.237,-64.689,-179.219,9.092,149.558
C05421=1110.417,175.988,-64.666,-179.221,9.089,149.558
C05422=1110.422,175.739,-64.642,-179.223,9.086,149.558
C05423=1110.426,175.491,-64.618,-179.225,9.083,149.558
C05424=1110.431,175.242,-64.595,-179.228,9.080,149.558
C05425=1110.435,174.993,-64.571,-179.229,9.077,149.558
C05426=1110.439,174.744,-64.547,-179.232,9.074,149.558
C05427=1110.444,174.495,-64.524,-179.234,9.071,149.558
C05428=1110.448,174.246,-64.500,-179.236,9.068,149.557
C05429=1110.452,174.033,-64.480,-179.238,9.065,149.557
C05430=1110.457,173.820,-64.459,-179.240,9.063,149.557
C05431=1110.461,173.606,-64.439,-179.242,9.061,149.557
C05432=1110.464,173.393,-64.420,-179.243,9.058,149.557
C05433=1110.468,173.180,-64.399,-179.245,9.056,149.557
C05434=1110.472,172.966,-64.379,-179.247,9.053,149.557
C05435=1110.476,172.753,-64.358,-179.249,9.051,149.557
C05436=1110.480,172.540,-64.338,-179.251,9.047,149.557
C05437=1110.484,172.291,-64.315,-179.253,9.045,149.557
C05438=1110.489,172.042,-64.292,-179.255,9.042,149.556
C05439=1110.493,171.793,-64.268,-179.258,9.039,149.556
C05440=1110.498,171.544,-64.244,-179.260,9.036,149.556
C05441=1110.503,171.295,-64.221,-179.262,9.033,149.556
C05442=1110.507,171.046,-64.198,-179.264,9.030,149.556
C05443=1110.511,170.798,-64.174,-179.266,9.027,149.556
C05444=1110.516,170.549,-64.151,-179.268,9.024,149.556
C05445=1110.521,170.300,-64.127,-179.271,9.021,149.556
C05446=1110.525,170.051,-64.104,-179.273,9.018,149.556
C05447=1110.530,169.802,-64.081,-179.275,9.015,149.556
C05448=1110.535,169.553,-64.057,-179.277,9.012,149.555
C05449=1110.539,169.304,-64.034,-179.279,9.009,149.555
C05450=1110.543,169.056,-64.010,-179.281,9.006,149.555
C05451=1110.548,168.807,-63.987,-179.284,9.003,149.555
C05452=1110.553,168.558,-63.964,-179.286,9.000,149.555
C05453=1110.558,168.309,-63.941,-179.288,8.997,149.555
C05454=1110.562,168.061,-63.918,-179.290,8.994,149.555
C05455=1110.566,167.812,-63.895,-179.292,8.990,149.555
C05456=1110.571,167.562,-63.871,-179.294,8.988,149.555
C05457=1110.576,167.313,-63.848,-179.297,8.985,149.555
C05458=1110.581,167.064,-63.824,-179.299,8.982,149.554
C05459=1110.585,166.816,-63.802,-179.301,8.979,149.554
C05460=1110.589,166.567,-63.778,-179.303,8.976,149.554
C05461=1110.594,166.318,-63.755,-179.305,8.973,149.554
C05462=1110.599,166.069,-63.732,-179.308,8.969,149.554
C05463=1110.603,165.821,-63.709,-179.309,8.967,149.554
C05464=1110.608,165.572,-63.686,-179.312,8.964,149.554
C05465=1110.613,165.323,-63.663,-179.314,8.960,149.553
C05466=1110.617,165.074,-63.640,-179.316,8.957,149.553
C05467=1110.621,164.825,-63.616,-179.318,8.955,149.553
C05468=1110.626,164.576,-63.593,-179.320,8.951,149.553
